LIN {X 0,Y 228.029,Z 967.337,A -85,B 0,C 180,E1 21811.233,E2 21811.233} C_VEL
LIN {X 0,Y 222.04,Z 977.557,A -85,B 0,C 180,E1 21813.343,E2 21813.343} C_VEL
LIN {X 0,Y 203.296,Z 1003.599,A -85,B 0,C 180,E1 21817.694,E2 21817.694} C_VEL
LIN {X 0,Y 184.311,Z 1025.745,A -85,B 0,C 180,E1 21824.225,E2 21824.225} C_VEL
LIN {X 0,Y 167.624,Z 1043.703,A -85,B 0,C 180,E1 21833.728,E2 21833.728} C_VEL
LIN {X 0,Y 157.775,Z 1054.755,A -85,B 0,C 180,E1 21844.418,E2 21844.418} C_VEL
LIN {X 0,Y 154.684,Z 1059.498,A -85,B 0,C 180,E1 21852.926,E2 21852.926} C_VEL
LIN {X 0,Y 154.96,Z 1063.359,A -85,B 0,C 180,E1 21867.202,E2 21867.202} C_VEL
LIN {X 0,Y 155.441,Z 1064.231,A -85,B 0,C 180,E1 21870.002,E2 21870.002} C_VEL
LIN {X 0,Y 154.103,Z 1063.62,A -85,B 0,C 180,E1 21881.334,E2 21881.334} C_VEL
LIN {X 0,Y 156.749,Z 1057.505,A -85,B 0,C 180,E1 21893.823,E2 21893.823} C_VEL
LIN {X 0,Y 166.557,Z 1045.003,A -85,B 0,C 180,E1 21905.9,E2 21905.9} C_VEL
LIN {X 0,Y 181.065,Z 1027.75,A -85,B 0,C 180,E1 21915.139,E2 21915.139} C_VEL
LIN {X 0,Y 197.137,Z 1006.697,A -85,B 0,C 180,E1 21921.789,E2 21921.789} C_VEL
LIN {X 0,Y 213.96,Z 980.35,A -85,B 0,C 180,E1 21926.713,E2 21926.713} C_VEL
LIN {X 0,Y 216.771,Z 975.207,A -85,B 0,C 180,E1 21927.424,E2 21927.424} C_VEL
LIN {X 0,Y 215.522,Z 959.866,A -85,B 0,C 180,E1 21933.374,E2 21933.374} C_VEL
LIN {X 0,Y 212.732,Z 946.935,A -85,B 0,C 180,E1 21940.342,E2 21940.342} C_VEL
LIN {X 0,Y 210.263,Z 938.618,A -85,B 0,C 180,E1 21947.476,E2 21947.476} C_VEL
LIN {X 0,Y 209.511,Z 933.278,A -85,B 0,C 180,E1 21955.804,E2 21955.804} C_VEL
LIN {X 0,Y 208.428,Z 937.644,A -85,B 0,C 180,E1 21964.111,E2 21964.111} C_VEL
LIN {X 0,Y 208.488,Z 945.436,A -85,B 0,C 180,E1 21971.461,E2 21971.461} C_VEL
LIN {X 0,Y 207.971,Z 957.227,A -85,B 0,C 180,E1 21978.834,E2 21978.834} C_VEL
LIN {X 0,Y 205.353,Z 971.666,A -85,B 0,C 180,E1 21986.184,E2 21986.184} C_VEL
LIN {X 0,Y 202.767,Z 979.395,A -85,B 0,C 180,E1 21989.847,E2 21989.847} C_VEL
LIN {X 0,Y 187.855,Z 996.811,A -85,B 0,C 180,E1 21996.292,E2 21996.292} C_VEL
LIN {X 0,Y 174.25,Z 1009.398,A -85,B 0,C 180,E1 22004.487,E2 22004.487} C_VEL
LIN {X 0,Y 164.735,Z 1016.233,A -85,B 0,C 180,E1 22013.313,E2 22013.313} C_VEL
LIN {X 0,Y 159.279,Z 1018.695,A -85,B 0,C 180,E1 22021.62,E2 22021.62} C_VEL
LIN {X 0,Y 156.492,Z 1018.02,A -85,B 0,C 180,E1 22029.898,E2 22029.898} C_VEL
LIN {X 0,Y 154.888,Z 1017.446,A -85,B 0,C 180,E1 22033.056,E2 22033.056} C_VEL
LIN {X 0,Y 149.377,Z 1013.798,A -85,B 0,C 180,E1 22041.859,E2 22041.859} C_VEL
LIN {X 0,Y 149.53,Z 1013.227,A -85,B 0,C 180,E1 22042.674,E2 22042.674} C_VEL
LIN {X 0,Y 155.199,Z 1001.57,A -85,B 0,C 180,E1 22054.194,E2 22054.194} C_VEL
LIN {X 0,Y 163.496,Z 986.022,A -85,B 0,C 180,E1 22063.22,E2 22063.22} C_VEL
LIN {X 0,Y 174.114,Z 964.454,A -85,B 0,C 180,E1 22071.019,E2 22071.019} C_VEL
LIN {X 0,Y 177.417,Z 956.35,A -85,B 0,C 180,E1 22073.245,E2 22073.245} C_VEL
LIN {X 0,Y 177.487,Z 938.518,A -85,B 0,C 180,E1 22079.2,E2 22079.2} C_VEL
LIN {X 0,Y 163.827,Z 940.595,A -85,B 0,C 180,E1 22083.878,E2 22083.878} C_VEL
LIN {X 0,Y 163.066,Z 940.258,A -85,B 0,C 180,E1 22084.495,E2 22084.495} C_VEL
LIN {X 0,Y 157.198,Z 966.499,A -85,B 0,C 180,E1 22090.811,E2 22090.811} C_VEL
LIN {X 0,Y 151.842,Z 988.828,A -85,B 0,C 180,E1 22099.154,E2 22099.154} C_VEL
LIN {X 0,Y 148.741,Z 1004.476,A -85,B 0,C 180,E1 22108.06,E2 22108.06} C_VEL
LIN {X 0,Y 148.185,Z 1016.057,A -85,B 0,C 180,E1 22118.312,E2 22118.312} C_VEL
LIN {X 0,Y 151.421,Z 1022.552,A -85,B 0,C 180,E1 22128.544,E2 22128.544} C_VEL
LIN {X 0,Y 155.312,Z 1024.197,A -85,B 0,C 180,E1 22134.48,E2 22134.48} C_VEL
LIN {X 0,Y 166.014,Z 1022.709,A -85,B 0,C 180,E1 22144.598,E2 22144.598} C_VEL
LIN {X 0,Y 180.205,Z 1015.966,A -85,B 0,C 180,E1 22153.03,E2 22153.03} C_VEL
LIN {X 0,Y 196.477,Z 1003.96,A -85,B 0,C 180,E1 22159.754,E2 22159.754} C_VEL
LIN {X 0,Y 214.009,Z 986.117,A -85,B 0,C 180,E1 22165.164,E2 22165.164} C_VEL
LIN {X 0,Y 220.51,Z 977.925,A -85,B 0,C 180,E1 22166.974,E2 22166.974} C_VEL
LIN {X 0,Y 222.968,Z 974.491,A -85,B 0,C 180,E1 22169.537,E2 22169.537} C_VEL
LIN {X 0,Y 222.507,Z 975.381,A -85,B 0,C 180,E1 22170.622,E2 22170.622} C_VEL
LIN {X 0,Y 215.741,Z 984.993,A -85,B 0,C 180,E1 22172.161,E2 22172.161} C_VEL
LIN {X 0,Y 194.53,Z 1010.583,A -85,B 0,C 180,E1 22177.084,E2 22177.084} C_VEL
LIN {X 0,Y 173.968,Z 1031.564,A -85,B 0,C 180,E1 22184.615,E2 22184.615} C_VEL
LIN {X 0,Y 157.729,Z 1046.889,A -85,B 0,C 180,E1 22194.836,E2 22194.836} C_VEL
LIN {X 0,Y 148.761,Z 1055.954,A -85,B 0,C 180,E1 22206.479,E2 22206.479} C_VEL
LIN {X 0,Y 146.505,Z 1059.588,A -85,B 0,C 180,E1 22218.074,E2 22218.074} C_VEL
LIN {X 0,Y 147.595,Z 1062.957,A -85,B 0,C 180,E1 22230.002,E2 22230.002} C_VEL
LIN {X 0,Y 146.253,Z 1062.469,A -85,B 0,C 180,E1 22241.952,E2 22241.952} C_VEL
LIN {X 0,Y 149.565,Z 1056.191,A -85,B 0,C 180,E1 22255.485,E2 22255.485} C_VEL
LIN {X 0,Y 160.402,Z 1043.804,A -85,B 0,C 180,E1 22267.849,E2 22267.849} C_VEL
LIN {X 0,Y 176.444,Z 1025.945,A -85,B 0,C 180,E1 22277.47,E2 22277.47} C_VEL
LIN {X 0,Y 193.605,Z 1004.417,A -85,B 0,C 180,E1 22284.083,E2 22284.083} C_VEL
LIN {X 0,Y 210.968,Z 977.854,A -85,B 0,C 180,E1 22288.843,E2 22288.843} C_VEL
LIN {X 0,Y 210.344,Z 964.721,A -85,B 0,C 180,E1 22294.366,E2 22294.366} C_VEL
LIN {X 0,Y 208.031,Z 951.826,A -85,B 0,C 180,E1 22301.908,E2 22301.908} C_VEL
LIN {X 0,Y 205.979,Z 944.435,A -85,B 0,C 180,E1 22309.361,E2 22309.361} C_VEL
LIN {X 0,Y 205.898,Z 940.4,A -85,B 0,C 180,E1 22315.731,E2 22315.731} C_VEL
LIN {X 0,Y 204.395,Z 944.731,A -85,B 0,C 180,E1 22324.192,E2 22324.192} C_VEL
LIN {X 0,Y 203.783,Z 952.605,A -85,B 0,C 180,E1 22331.683,E2 22331.683} C_VEL
LIN {X 0,Y 202.215,Z 964.628,A -85,B 0,C 180,E1 22339.392,E2 22339.392} C_VEL
LIN {X 0,Y 198.723,Z 977.474,A -85,B 0,C 180,E1 22346.237,E2 22346.237} C_VEL
LIN {X 0,Y 195.713,Z 983.429,A -85,B 0,C 180,E1 22348.932,E2 22348.932} C_VEL
LIN {X 0,Y 179.086,Z 1001.128,A -85,B 0,C 180,E1 22356.191,E2 22356.191} C_VEL
LIN {X 0,Y 165.411,Z 1012.493,A -85,B 0,C 180,E1 22364.814,E2 22364.814} C_VEL
LIN {X 0,Y 155.851,Z 1018.408,A -85,B 0,C 180,E1 22374.343,E2 22374.343} C_VEL
LIN {X 0,Y 149.602,Z 1019.899,A -85,B 0,C 180,E1 22386.117,E2 22386.117} C_VEL
LIN {X 0,Y 148.554,Z 1016.055,A -85,B 0,C 180,E1 22398.236,E2 22398.236} C_VEL
LIN {X 0,Y 149.53,Z 1013.227,A -85,B 0,C 180,E1 22402.674,E2 22402.674} C_VEL
LIN {X 0,Y 148.875,Z 1009.687,A -85,B 0,C 180,E1 22407.527,E2 22407.527} C_VEL
LIN {X 0,Y 147.619,Z 1003.02,A -85,B 0,C 180,E1 22414.754,E2 22414.754} C_VEL
LIN {X 0,Y 148.064,Z 1002.082,A -85,B 0,C 180,E1 22415.512,E2 22415.512} C_VEL
LIN {X 0,Y 157.724,Z 984.901,A -85,B 0,C 180,E1 22425.507,E2 22425.507} C_VEL
LIN {X 0,Y 168.707,Z 963.403,A -85,B 0,C 180,E1 22433.117,E2 22433.117} C_VEL
LIN {X 0,Y 170.899,Z 957.374,A -85,B 0,C 180,E1 22434.885,E2 22434.885} C_VEL
LIN {X 0,Y 170.904,Z 945.87,A -85,B 0,C 180,E1 22439.151,E2 22439.151} C_VEL
LIN {X 0,Y 161.241,Z 947.296,A -85,B 0,C 180,E1 22442.484,E2 22442.484} C_VEL
LIN {X 0,Y 155.877,Z 949.306,A -85,B 0,C 180,E1 22444.086,E2 22444.086} C_VEL
LIN {X 0,Y 153.649,Z 949.749,A -85,B 0,C 180,E1 22445.448,E2 22445.448} C_VEL
LIN {X 0,Y 147.267,Z 975.851,A -85,B 0,C 180,E1 22453.042,E2 22453.042} C_VEL
LIN {X 0,Y 142.62,Z 995.639,A -85,B 0,C 180,E1 22462.03,E2 22462.03} C_VEL
LIN {X 0,Y 140.25,Z 1010.132,A -85,B 0,C 180,E1 22472.02,E2 22472.02} C_VEL
LIN {X 0,Y 141.614,Z 1020.907,A -85,B 0,C 180,E1 22484.197,E2 22484.197} C_VEL
LIN {X 0,Y 146.983,Z 1025.26,A -85,B 0,C 180,E1 22494.166,E2 22494.166} C_VEL
LIN {X 0,Y 152.277,Z 1025.845,A -85,B 0,C 180,E1 22500.073,E2 22500.073} C_VEL
LIN {X 0,Y 166.607,Z 1022.246,A -85,B 0,C 180,E1 22510.535,E2 22510.535} C_VEL
LIN {X 0,Y 183.215,Z 1013.219,A -85,B 0,C 180,E1 22518.318,E2 22518.318} C_VEL
LIN {X 0,Y 202.615,Z 997.714,A -85,B 0,C 180,E1 22524.712,E2 22524.712} C_VEL
LIN {X 0,Y 216.289,Z 983.083,A -85,B 0,C 180,E1 22528.243,E2 22528.243} C_VEL
LIN {X 0,Y 217.862,Z 981.272,A -85,B 0,C 180,E1 22529.154,E2 22529.154} C_VEL
LIN {X 0,Y 216.382,Z 983.183,A -85,B 0,C 180,E1 22529.731,E2 22529.731} C_VEL
LIN {X 0,Y 194.367,Z 1008.192,A -85,B 0,C 180,E1 22534.143,E2 22534.143} C_VEL
LIN {X 0,Y 172.775,Z 1028.508,A -85,B 0,C 180,E1 22540.887,E2 22540.887} C_VEL
LIN {X 0,Y 154.561,Z 1043.785,A -85,B 0,C 180,E1 22550.453,E2 22550.453} C_VEL
LIN {X 0,Y 143.327,Z 1053.143,A -85,B 0,C 180,E1 22561.619,E2 22561.619} C_VEL
LIN {X 0,Y 139.345,Z 1057.074,A -85,B 0,C 180,E1 22570.978,E2 22570.978} C_VEL
LIN {X 0,Y 138.869,Z 1058.428,A -85,B 0,C 180,E1 22581.609,E2 22581.609} C_VEL
LIN {X 0,Y 139.755,Z 1061.663,A -85,B 0,C 180,E1 22590.002,E2 22590.002} C_VEL
LIN {X 0,Y 138.392,Z 1061.312,A -85,B 0,C 180,E1 22602.641,E2 22602.641} C_VEL
LIN {X 0,Y 142.279,Z 1055.149,A -85,B 0,C 180,E1 22616.892,E2 22616.892} C_VEL
LIN {X 0,Y 154.065,Z 1042.938,A -85,B 0,C 180,E1 22629.704,E2 22629.704} C_VEL
LIN {X 0,Y 170.283,Z 1026.144,A -85,B 0,C 180,E1 22639.096,E2 22639.096} C_VEL
LIN {X 0,Y 189.151,Z 1003.779,A -85,B 0,C 180,E1 22646.081,E2 22646.081} C_VEL
LIN {X 0,Y 205.232,Z 980.507,A -85,B 0,C 180,E1 22650.343,E2 22650.343} C_VEL
LIN {X 0,Y 204.846,Z 967.229,A -85,B 0,C 180,E1 22656.543,E2 22656.543} C_VEL
LIN {X 0,Y 203.246,Z 956.398,A -85,B 0,C 180,E1 22663.73,E2 22663.73} C_VEL
LIN {X 0,Y 201.732,Z 950.029,A -85,B 0,C 180,E1 22671.315,E2 22671.315} C_VEL
LIN {X 0,Y 201.977,Z 947.406,A -85,B 0,C 180,E1 22675.648,E2 22675.648} C_VEL
LIN {X 0,Y 200.398,Z 950.179,A -85,B 0,C 180,E1 22682.109,E2 22682.109} C_VEL
LIN {X 0,Y 199.376,Z 956.143,A -85,B 0,C 180,E1 22689.157,E2 22689.157} C_VEL
LIN {X 0,Y 197.202,Z 967.09,A -85,B 0,C 180,E1 22697.111,E2 22697.111} C_VEL
LIN {X 0,Y 193.399,Z 979.33,A -85,B 0,C 180,E1 22704.201,E2 22704.201} C_VEL
LIN {X 0,Y 191.142,Z 984.423,A -85,B 0,C 180,E1 22706.977,E2 22706.977} C_VEL
LIN {X 0,Y 174.334,Z 1001.641,A -85,B 0,C 180,E1 22713.998,E2 22713.998} C_VEL
LIN {X 0,Y 159.666,Z 1013.238,A -85,B 0,C 180,E1 22722.697,E2 22722.697} C_VEL
LIN {X 0,Y 149.196,Z 1019.423,A -85,B 0,C 180,E1 22732.488,E2 22732.488} C_VEL
LIN {X 0,Y 142.17,Z 1021.163,A -85,B 0,C 180,E1 22744.784,E2 22744.784} C_VEL
LIN {X 0,Y 140.634,Z 1017.58,A -85,B 0,C 180,E1 22757.563,E2 22757.563} C_VEL
LIN {X 0,Y 144.696,Z 1008.44,A -85,B 0,C 180,E1 22769.998,E2 22769.998} C_VEL
LIN {X 0,Y 148.064,Z 1002.082,A -85,B 0,C 180,E1 22775.512,E2 22775.512} C_VEL
LIN {X 0,Y 147.385,Z 997.386,A -85,B 0,C 180,E1 22779.727,E2 22779.727} C_VEL
LIN {X 0,Y 147.297,Z 992.02,A -85,B 0,C 180,E1 22783.836,E2 22783.836} C_VEL
LIN {X 0,Y 158.653,Z 971.863,A -85,B 0,C 180,E1 22792.439,E2 22792.439} C_VEL
LIN {X 0,Y 164.249,Z 960.2,A -85,B 0,C 180,E1 22795.966,E2 22795.966} C_VEL
LIN {X 0,Y 165.075,Z 952.705,A -85,B 0,C 180,E1 22798.78,E2 22798.78} C_VEL
LIN {X 0,Y 152.734,Z 955.58,A -85,B 0,C 180,E1 22802.756,E2 22802.756} C_VEL
LIN {X 0,Y 145.006,Z 957.339,A -85,B 0,C 180,E1 22805.811,E2 22805.811} C_VEL
LIN {X 0,Y 143.906,Z 959.455,A -85,B 0,C 180,E1 22806.868,E2 22806.868} C_VEL
LIN {X 0,Y 137.626,Z 983.982,A -85,B 0,C 180,E1 22815.55,E2 22815.55} C_VEL
LIN {X 0,Y 133.503,Z 1002.243,A -85,B 0,C 180,E1 22825.573,E2 22825.573} C_VEL
LIN {X 0,Y 132.268,Z 1015.032,A -85,B 0,C 180,E1 22836.309,E2 22836.309} C_VEL
LIN {X 0,Y 134.774,Z 1023.078,A -85,B 0,C 180,E1 22847.106,E2 22847.106} C_VEL
LIN {X 0,Y 138.569,Z 1026.061,A -85,B 0,C 180,E1 22853.81,E2 22853.81} C_VEL
LIN {X 0,Y 150.685,Z 1026.951,A -85,B 0,C 180,E1 22865.838,E2 22865.838} C_VEL
LIN {X 0,Y 165.335,Z 1022.545,A -85,B 0,C 180,E1 22874.598,E2 22874.598} C_VEL
LIN {X 0,Y 183.447,Z 1012.761,A -85,B 0,C 180,E1 22881.858,E2 22881.858} C_VEL
LIN {X 0,Y 202.545,Z 997.761,A -85,B 0,C 180,E1 22887.41,E2 22887.41} C_VEL
LIN {X 0,Y 207.432,Z 993.164,A -85,B 0,C 180,E1 22888.851,E2 22888.851} C_VEL
LIN {X 0,Y 182.769,Z 1016.977,A -85,B 0,C 180,E1 22894.067,E2 22894.067} C_VEL
LIN {X 0,Y 161.491,Z 1034.127,A -85,B 0,C 180,E1 22901.408,E2 22901.408} C_VEL
LIN {X 0,Y 143.469,Z 1047.146,A -85,B 0,C 180,E1 22912.252,E2 22912.252} C_VEL
LIN {X 0,Y 133.19,Z 1054.601,A -85,B 0,C 180,E1 22925.572,E2 22925.572} C_VEL
LIN {X 0,Y 131.057,Z 1057.283,A -85,B 0,C 180,E1 22941.64,E2 22941.64} C_VEL
LIN {X 0,Y 131.933,Z 1060.373,A -85,B 0,C 180,E1 22950.002,E2 22950.002} C_VEL
LIN {X 0,Y 130.575,Z 1060.156,A -85,B 0,C 180,E1 22963.412,E2 22963.412} C_VEL
LIN {X 0,Y 134.172,Z 1055.063,A -85,B 0,C 180,E1 22976.835,E2 22976.835} C_VEL
LIN {X 0,Y 146.125,Z 1043.754,A -85,B 0,C 180,E1 22990.363,E2 22990.363} C_VEL
LIN {X 0,Y 163.909,Z 1026.724,A -85,B 0,C 180,E1 23000.683,E2 23000.683} C_VEL
LIN {X 0,Y 183.386,Z 1005.118,A -85,B 0,C 180,E1 23007.733,E2 23007.733} C_VEL
LIN {X 0,Y 199.357,Z 983.496,A -85,B 0,C 180,E1 23011.835,E2 23011.835} C_VEL
LIN {X 0,Y 199.558,Z 971.859,A -85,B 0,C 180,E1 23017.656,E2 23017.656} C_VEL
LIN {X 0,Y 198.579,Z 962.28,A -85,B 0,C 180,E1 23024.471,E2 23024.471} C_VEL
LIN {X 0,Y 197.643,Z 954.687,A -85,B 0,C 180,E1 23034.82,E2 23034.82} C_VEL
LIN {X 0,Y 196.526,Z 955.593,A -85,B 0,C 180,E1 23039.944,E2 23039.944} C_VEL
LIN {X 0,Y 194.441,Z 962.436,A -85,B 0,C 180,E1 23048.898,E2 23048.898} C_VEL
LIN {X 0,Y 191.799,Z 971.74,A -85,B 0,C 180,E1 23056.094,E2 23056.094} C_VEL
LIN {X 0,Y 187.488,Z 982.869,A -85,B 0,C 180,E1 23063.042,E2 23063.042} C_VEL
LIN {X 0,Y 184.832,Z 987.642,A -85,B 0,C 180,E1 23065.695,E2 23065.695} C_VEL
LIN {X 0,Y 166.835,Z 1004.649,A -85,B 0,C 180,E1 23073.103,E2 23073.103} C_VEL
LIN {X 0,Y 150.501,Z 1016.3,A -85,B 0,C 180,E1 23083.163,E2 23083.163} C_VEL
LIN {X 0,Y 142.725,Z 1020.435,A -85,B 0,C 180,E1 23090.466,E2 23090.466} C_VEL
LIN {X 0,Y 134.571,Z 1022.36,A -85,B 0,C 180,E1 23103.931,E2 23103.931} C_VEL
LIN {X 0,Y 132.751,Z 1019.042,A -85,B 0,C 180,E1 23116.812,E2 23116.812} C_VEL
LIN {X 0,Y 136.703,Z 1010.183,A -85,B 0,C 180,E1 23129.998,E2 23129.998} C_VEL
LIN {X 0,Y 144.762,Z 996.321,A -85,B 0,C 180,E1 23141.307,E2 23141.307} C_VEL
LIN {X 0,Y 147.297,Z 992.02,A -85,B 0,C 180,E1 23143.836,E2 23143.836} C_VEL
LIN {X 0,Y 149.883,Z 982.506,A -85,B 0,C 180,E1 23149.419,E2 23149.419} C_VEL
LIN {X 0,Y 152.958,Z 971.748,A -85,B 0,C 180,E1 23154.546,E2 23154.546} C_VEL
LIN {X 0,Y 158.067,Z 960.594,A -85,B 0,C 180,E1 23158.117,E2 23158.117} C_VEL
LIN {X 0,Y 158.278,Z 959.448,A -85,B 0,C 180,E1 23158.572,E2 23158.572} C_VEL
LIN {X 0,Y 138.692,Z 964.583,A -85,B 0,C 180,E1 23165.213,E2 23165.213} C_VEL
LIN {X 0,Y 134.955,Z 965.203,A -85,B 0,C 180,E1 23167.555,E2 23167.555} C_VEL
LIN {X 0,Y 128.999,Z 987.722,A -85,B 0,C 180,E1 23176.536,E2 23176.536} C_VEL
LIN {X 0,Y 124.976,Z 1006.133,A -85,B 0,C 180,E1 23187.996,E2 23187.996} C_VEL
LIN {X 0,Y 124.791,Z 1018.676,A -85,B 0,C 180,E1 23200.228,E2 23200.228} C_VEL
LIN {X 0,Y 130.146,Z 1026.576,A -85,B 0,C 180,E1 23213.408,E2 23213.408} C_VEL
LIN {X 0,Y 142.495,Z 1028.813,A -85,B 0,C 180,E1 23226.175,E2 23226.175} C_VEL
LIN {X 0,Y 156.657,Z 1025.904,A -85,B 0,C 180,E1 23234.882,E2 23234.882} C_VEL
LIN {X 0,Y 176.323,Z 1017.193,A -85,B 0,C 180,E1 23242.854,E2 23242.854} C_VEL
LIN {X 0,Y 195.416,Z 1004.39,A -85,B 0,C 180,E1 23248.282,E2 23248.282} C_VEL
LIN {X 0,Y 168.399,Z 1026.15,A -85,B 0,C 180,E1 23254.875,E2 23254.875} C_VEL
LIN {X 0,Y 146.792,Z 1040.697,A -85,B 0,C 180,E1 23263.782,E2 23263.782} C_VEL
LIN {X 0,Y 131.981,Z 1049.734,A -85,B 0,C 180,E1 23275.001,E2 23275.001} C_VEL
LIN {X 0,Y 124.221,Z 1054.414,A -85,B 0,C 180,E1 23288.555,E2 23288.555} C_VEL
LIN {X 0,Y 123.246,Z 1055.205,A -85,B 0,C 180,E1 23299.72,E2 23299.72} C_VEL
LIN {X 0,Y 124.106,Z 1059.083,A -85,B 0,C 180,E1 23310.002,E2 23310.002} C_VEL
LIN {X 0,Y 122.766,Z 1058.971,A -85,B 0,C 180,E1 23324.283,E2 23324.283} C_VEL
LIN {X 0,Y 126.979,Z 1054.032,A -85,B 0,C 180,E1 23338.489,E2 23338.489} C_VEL
LIN {X 0,Y 140.052,Z 1042.895,A -85,B 0,C 180,E1 23352.51,E2 23352.51} C_VEL
LIN {X 0,Y 158.931,Z 1026.054,A -85,B 0,C 180,E1 23362.929,E2 23362.929} C_VEL
LIN {X 0,Y 179.345,Z 1004.546,A -85,B 0,C 180,E1 23369.924,E2 23369.924} C_VEL
LIN {X 0,Y 193.251,Z 986.794,A -85,B 0,C 180,E1 23373.352,E2 23373.352} C_VEL
LIN {X 0,Y 194.165,Z 978.377,A -85,B 0,C 180,E1 23377.606,E2 23377.606} C_VEL
LIN {X 0,Y 193.709,Z 968.016,A -85,B 0,C 180,E1 23385.231,E2 23385.231} C_VEL
LIN {X 0,Y 193.253,Z 960.939,A -85,B 0,C 180,E1 23395.451,E2 23395.451} C_VEL
LIN {X 0,Y 191.151,Z 963.426,A -85,B 0,C 180,E1 23402.211,E2 23402.211} C_VEL
LIN {X 0,Y 189.072,Z 969.071,A -85,B 0,C 180,E1 23409.153,E2 23409.153} C_VEL
LIN {X 0,Y 185.44,Z 978.512,A -85,B 0,C 180,E1 23416.661,E2 23416.661} C_VEL
LIN {X 0,Y 179.534,Z 989.844,A -85,B 0,C 180,E1 23423.956,E2 23423.956} C_VEL
LIN {X 0,Y 161.766,Z 1005.771,A -85,B 0,C 180,E1 23430.995,E2 23430.995} C_VEL
LIN {X 0,Y 144.843,Z 1017.198,A -85,B 0,C 180,E1 23440.853,E2 23440.853} C_VEL
LIN {X 0,Y 132.538,Z 1022.819,A -85,B 0,C 180,E1 23452.925,E2 23452.925} C_VEL
LIN {X 0,Y 127.549,Z 1023.61,A -85,B 0,C 180,E1 23461.649,E2 23461.649} C_VEL
LIN {X 0,Y 124.867,Z 1020.5,A -85,B 0,C 180,E1 23475.963,E2 23475.963} C_VEL
LIN {X 0,Y 128.692,Z 1011.925,A -85,B 0,C 180,E1 23489.998,E2 23489.998} C_VEL
LIN {X 0,Y 137.734,Z 997.286,A -85,B 0,C 180,E1 23502.698,E2 23502.698} C_VEL
LIN {X 0,Y 149.459,Z 977.971,A -85,B 0,C 180,E1 23512.325,E2 23512.325} C_VEL
LIN {X 0,Y 152.958,Z 971.748,A -85,B 0,C 180,E1 23514.546,E2 23514.546} C_VEL
LIN {X 0,Y 152.567,Z 968.801,A -85,B 0,C 180,E1 23516.328,E2 23516.328} C_VEL
LIN {X 0,Y 146.457,Z 967.65,A -85,B 0,C 180,E1 23519.581,E2 23519.581} C_VEL
LIN {X 0,Y 130.899,Z 971.037,A -85,B 0,C 180,E1 23525.587,E2 23525.587} C_VEL
LIN {X 0,Y 125.47,Z 972.244,A -85,B 0,C 180,E1 23528.957,E2 23528.957} C_VEL
LIN {X 0,Y 119.632,Z 994.25,A -85,B 0,C 180,E1 23539.404,E2 23539.404} C_VEL
LIN {X 0,Y 116.541,Z 1011.595,A -85,B 0,C 180,E1 23552.413,E2 23552.413} C_VEL
LIN {X 0,Y 118.821,Z 1023.708,A -85,B 0,C 180,E1 23567.217,E2 23567.217} C_VEL
LIN {X 0,Y 127.173,Z 1029.413,A -85,B 0,C 180,E1 23580.087,E2 23580.087} C_VEL
LIN {X 0,Y 142.698,Z 1029.846,A -85,B 0,C 180,E1 23592.326,E2 23592.326} C_VEL
LIN {X 0,Y 163.175,Z 1023.959,A -85,B 0,C 180,E1 23601.85,E2 23601.85} C_VEL
LIN {X 0,Y 182.474,Z 1014.154,A -85,B 0,C 180,E1 23607.808,E2 23607.808} C_VEL
LIN {X 0,Y 154.125,Z 1033.298,A -85,B 0,C 180,E1 23615.863,E2 23615.863} C_VEL
LIN {X 0,Y 132.618,Z 1045.282,A -85,B 0,C 180,E1 23626.767,E2 23626.767} C_VEL
LIN {X 0,Y 120.089,Z 1051.454,A -85,B 0,C 180,E1 23639.717,E2 23639.717} C_VEL
LIN {X 0,Y 115.435,Z 1053.768,A -85,B 0,C 180,E1 23659.016,E2 23659.016} C_VEL
LIN {X 0,Y 116.243,Z 1057.776,A -85,B 0,C 180,E1 23670.003,E2 23670.003} C_VEL
LIN {X 0,Y 114.997,Z 1057.775,A -85,B 0,C 180,E1 23685.27,E2 23685.27} C_VEL
LIN {X 0,Y 119.913,Z 1053.002,A -85,B 0,C 180,E1 23700.338,E2 23700.338} C_VEL
LIN {X 0,Y 134.183,Z 1042.019,A -85,B 0,C 180,E1 23714.851,E2 23714.851} C_VEL
LIN {X 0,Y 154.189,Z 1025.383,A -85,B 0,C 180,E1 23725.328,E2 23725.328} C_VEL
LIN {X 0,Y 175.46,Z 1004.082,A -85,B 0,C 180,E1 23732.193,E2 23732.193} C_VEL
LIN {X 0,Y 187.382,Z 989.809,A -85,B 0,C 180,E1 23734.984,E2 23734.984} C_VEL
LIN {X 0,Y 188.486,Z 984.741,A -85,B 0,C 180,E1 23737.484,E2 23737.484} C_VEL
LIN {X 0,Y 188.712,Z 975.319,A -85,B 0,C 180,E1 23744.326,E2 23744.326} C_VEL
LIN {X 0,Y 188.227,Z 968.687,A -85,B 0,C 180,E1 23753.014,E2 23753.014} C_VEL
LIN {X 0,Y 188.466,Z 967.417,A -85,B 0,C 180,E1 23755.335,E2 23755.335} C_VEL
LIN {X 0,Y 186.092,Z 969.785,A -85,B 0,C 180,E1 23762.271,E2 23762.271} C_VEL
LIN {X 0,Y 183.359,Z 975.524,A -85,B 0,C 180,E1 23769.44,E2 23769.44} C_VEL
LIN {X 0,Y 178.75,Z 984.72,A -85,B 0,C 180,E1 23776.936,E2 23776.936} C_VEL
LIN {X 0,Y 174.361,Z 991.929,A -85,B 0,C 180,E1 23781.92,E2 23781.92} C_VEL
LIN {X 0,Y 156.033,Z 1007.554,A -85,B 0,C 180,E1 23789.149,E2 23789.149} C_VEL
LIN {X 0,Y 137.652,Z 1019.046,A -85,B 0,C 180,E1 23799.647,E2 23799.647} C_VEL
LIN {X 0,Y 124.62,Z 1024.269,A -85,B 0,C 180,E1 23812.589,E2 23812.589} C_VEL
LIN {X 0,Y 117.791,Z 1024.046,A -85,B 0,C 180,E1 23827.315,E2 23827.315} C_VEL
LIN {X 0,Y 118,Z 1018.524,A -85,B 0,C 180,E1 23842.625,E2 23842.625} C_VEL
LIN {X 0,Y 124.668,Z 1007.356,A -85,B 0,C 180,E1 23856.973,E2 23856.973} C_VEL
LIN {X 0,Y 135.492,Z 991.218,A -85,B 0,C 180,E1 23868.472,E2 23868.472} C_VEL
LIN {X 0,Y 148.358,Z 970.014,A -85,B 0,C 180,E1 23877.319,E2 23877.319} C_VEL
LIN {X 0,Y 150.004,Z 967.156,A -85,B 0,C 180,E1 23878.192,E2 23878.192} C_VEL
LIN {X 0,Y 147.276,Z 967.341,A -85,B 0,C 180,E1 23879.29,E2 23879.29} C_VEL
LIN {X 0,Y 130.899,Z 971.037,A -85,B 0,C 180,E1 23885.587,E2 23885.587} C_VEL
LIN {X 0,Y 121.588,Z 975.266,A -85,B 0,C 180,E1 23888.718,E2 23888.718} C_VEL
LIN {X 0,Y 115.514,Z 980.97,A -85,B 0,C 180,E1 23891.588,E2 23891.588} C_VEL
LIN {X 0,Y 115.134,Z 981.973,A -85,B 0,C 180,E1 23892.078,E2 23892.078} C_VEL
LIN {X 0,Y 110.009,Z 1002.178,A -85,B 0,C 180,E1 23904.191,E2 23904.191} C_VEL
LIN {X 0,Y 108.657,Z 1016.609,A -85,B 0,C 180,E1 23917.589,E2 23917.589} C_VEL
LIN {X 0,Y 113.236,Z 1026.743,A -85,B 0,C 180,E1 23932.418,E2 23932.418} C_VEL
LIN {X 0,Y 125.938,Z 1031.738,A -85,B 0,C 180,E1 23946.991,E2 23946.991} C_VEL
LIN {X 0,Y 144.626,Z 1030.42,A -85,B 0,C 180,E1 23958.377,E2 23958.377} C_VEL
LIN {X 0,Y 165.119,Z 1023.926,A -85,B 0,C 180,E1 23966.072,E2 23966.072} C_VEL
LIN {X 0,Y 169.419,Z 1022.041,A -85,B 0,C 180,E1 23967.318,E2 23967.318} C_VEL
LIN {X 0,Y 163.822,Z 1025.642,A -85,B 0,C 180,E1 23969.215,E2 23969.215} C_VEL
LIN {X 0,Y 138.347,Z 1039.394,A -85,B 0,C 180,E1 23977.896,E2 23977.896} C_VEL
LIN {X 0,Y 119.101,Z 1047.95,A -85,B 0,C 180,E1 23990.537,E2 23990.537} C_VEL
LIN {X 0,Y 109.428,Z 1051.458,A -85,B 0,C 180,E1 24005.478,E2 24005.478} C_VEL
LIN {X 0,Y 107.767,Z 1051.574,A -85,B 0,C 180,E1 24016.712,E2 24016.712} C_VEL
LIN {X 0,Y 108.404,Z 1056.474,A -85,B 0,C 180,E1 24030.003,E2 24030.003} C_VEL
LIN {X 0,Y 107.267,Z 1056.579,A -85,B 0,C 180,E1 24046.401,E2 24046.401} C_VEL
LIN {X 0,Y 112.983,Z 1051.962,A -85,B 0,C 180,E1 24062.418,E2 24062.418} C_VEL
LIN {X 0,Y 128.542,Z 1041.143,A -85,B 0,C 180,E1 24077.41,E2 24077.41} C_VEL
LIN {X 0,Y 149.758,Z 1024.705,A -85,B 0,C 180,E1 24087.861,E2 24087.861} C_VEL
LIN {X 0,Y 171.866,Z 1003.618,A -85,B 0,C 180,E1 24094.558,E2 24094.558} C_VEL
LIN {X 0,Y 182.432,Z 991.181,A -85,B 0,C 180,E1 24097.165,E2 24097.165} C_VEL
LIN {X 0,Y 183.332,Z 981.954,A -85,B 0,C 180,E1 24103.853,E2 24103.853} C_VEL
LIN {X 0,Y 183.166,Z 976.388,A -85,B 0,C 180,E1 24110.427,E2 24110.427} C_VEL
LIN {X 0,Y 183.409,Z 973.696,A -85,B 0,C 180,E1 24115.206,E2 24115.206} C_VEL
LIN {X 0,Y 180.871,Z 975.793,A -85,B 0,C 180,E1 24122.096,E2 24122.096} C_VEL
LIN {X 0,Y 177.263,Z 981.814,A -85,B 0,C 180,E1 24129.768,E2 24129.768} C_VEL
LIN {X 0,Y 172.484,Z 989.573,A -85,B 0,C 180,E1 24136.377,E2 24136.377} C_VEL
LIN {X 0,Y 168.492,Z 995.06,A -85,B 0,C 180,E1 24140.445,E2 24140.445} C_VEL
LIN {X 0,Y 149.494,Z 1010.031,A -85,B 0,C 180,E1 24147.596,E2 24147.596} C_VEL
LIN {X 0,Y 132.523,Z 1019.881,A -85,B 0,C 180,E1 24156.89,E2 24156.89} C_VEL
LIN {X 0,Y 118.163,Z 1025.352,A -85,B 0,C 180,E1 24170.155,E2 24170.155} C_VEL
LIN {X 0,Y 110.314,Z 1025.367,A -85,B 0,C 180,E1 24185.682,E2 24185.682} C_VEL
LIN {X 0,Y 109.993,Z 1020.105,A -85,B 0,C 180,E1 24202.085,E2 24202.085} C_VEL
LIN {X 0,Y 116.785,Z 1009.231,A -85,B 0,C 180,E1 24217.447,E2 24217.447} C_VEL
LIN {X 0,Y 127.684,Z 993.905,A -85,B 0,C 180,E1 24229.371,E2 24229.371} C_VEL
LIN {X 0,Y 139.59,Z 975.829,A -85,B 0,C 180,E1 24237.687,E2 24237.687} C_VEL
LIN {X 0,Y 139.929,Z 974.072,A -85,B 0,C 180,E1 24238.673,E2 24238.673} C_VEL
LIN {X 0,Y 116.078,Z 978.546,A -85,B 0,C 180,E1 24250.501,E2 24250.501} C_VEL
LIN {X 0,Y 115.134,Z 981.973,A -85,B 0,C 180,E1 24252.078,E2 24252.078} C_VEL
LIN {X 0,Y 110.282,Z 990.768,A -85,B 0,C 180,E1 24256.428,E2 24256.428} C_VEL
LIN {X 0,Y 102.196,Z 1002.375,A -85,B 0,C 180,E1 24263.966,E2 24263.966} C_VEL
LIN {X 0,Y 101.873,Z 1003.631,A -85,B 0,C 180,E1 24264.96,E2 24264.96} C_VEL
LIN {X 0,Y 101.161,Z 1019.001,A -85,B 0,C 180,E1 24280.728,E2 24280.728} C_VEL
LIN {X 0,Y 108.188,Z 1029.283,A -85,B 0,C 180,E1 24297.505,E2 24297.505} C_VEL
LIN {X 0,Y 123.934,Z 1033.464,A -85,B 0,C 180,E1 24312.23,E2 24312.23} C_VEL
LIN {X 0,Y 142.482,Z 1031.901,A -85,B 0,C 180,E1 24321.908,E2 24321.908} C_VEL
LIN {X 0,Y 156.202,Z 1028.324,A -85,B 0,C 180,E1 24326.81,E2 24326.81} C_VEL
LIN {X 0,Y 156.491,Z 1028.472,A -85,B 0,C 180,E1 24327.653,E2 24327.653} C_VEL
LIN {X 0,Y 128.702,Z 1041.222,A -85,B 0,C 180,E1 24337.435,E2 24337.435} C_VEL
LIN {X 0,Y 112.997,Z 1046.956,A -85,B 0,C 180,E1 24347.94,E2 24347.94} C_VEL
LIN {X 0,Y 102.193,Z 1049.828,A -85,B 0,C 180,E1 24363.614,E2 24363.614} C_VEL
LIN {X 0,Y 100.175,Z 1049.615,A -85,B 0,C 180,E1 24374.666,E2 24374.666} C_VEL
LIN {X 0,Y 100.533,Z 1055.17,A -85,B 0,C 180,E1 24390.003,E2 24390.003} C_VEL
LIN {X 0,Y 99.571,Z 1055.383,A -85,B 0,C 180,E1 24407.708,E2 24407.708} C_VEL
LIN {X 0,Y 106.235,Z 1050.902,A -85,B 0,C 180,E1 24424.76,E2 24424.76} C_VEL
LIN {X 0,Y 123.188,Z 1040.266,A -85,B 0,C 180,E1 24440.194,E2 24440.194} C_VEL
LIN {X 0,Y 145.637,Z 1024.026,A -85,B 0,C 180,E1 24450.543,E2 24450.543} C_VEL
LIN {X 0,Y 168.504,Z 1003.238,A -85,B 0,C 180,E1 24456.998,E2 24456.998} C_VEL
LIN {X 0,Y 176.017,Z 995.208,A -85,B 0,C 180,E1 24458.576,E2 24458.576} C_VEL
LIN {X 0,Y 177.614,Z 987.993,A -85,B 0,C 180,E1 24463.746,E2 24463.746} C_VEL
LIN {X 0,Y 177.823,Z 982.505,A -85,B 0,C 180,E1 24470.136,E2 24470.136} C_VEL
LIN {X 0,Y 178.092,Z 979.771,A -85,B 0,C 180,E1 24475.063,E2 24475.063} C_VEL
LIN {X 0,Y 175.146,Z 981.901,A -85,B 0,C 180,E1 24482.413,E2 24482.413} C_VEL
LIN {X 0,Y 170.786,Z 987.911,A -85,B 0,C 180,E1 24490.142,E2 24490.142} C_VEL
LIN {X 0,Y 164.075,Z 996.63,A -85,B 0,C 180,E1 24497.733,E2 24497.733} C_VEL
LIN {X 0,Y 160.56,Z 999.903,A -85,B 0,C 180,E1 24499.433,E2 24499.433} C_VEL
LIN {X 0,Y 139.961,Z 1014.296,A -85,B 0,C 180,E1 24507.307,E2 24507.307} C_VEL
LIN {X 0,Y 121.34,Z 1023.485,A -85,B 0,C 180,E1 24518.465,E2 24518.465} C_VEL
LIN {X 0,Y 111.979,Z 1026.434,A -85,B 0,C 180,E1 24527.46,E2 24527.46} C_VEL
LIN {X 0,Y 102.944,Z 1026.693,A -85,B 0,C 180,E1 24543.814,E2 24543.814} C_VEL
LIN {X 0,Y 101.99,Z 1021.679,A -85,B 0,C 180,E1 24561.46,E2 24561.46} C_VEL
LIN {X 0,Y 108.897,Z 1011.081,A -85,B 0,C 180,E1 24577.989,E2 24577.989} C_VEL
LIN {X 0,Y 120.843,Z 995.291,A -85,B 0,C 180,E1 24591.111,E2 24591.111} C_VEL
LIN {X 0,Y 130.928,Z 981.073,A -85,B 0,C 180,E1 24598.224,E2 24598.224} C_VEL
LIN {X 0,Y 123.96,Z 981.85,A -85,B 0,C 180,E1 24601.453,E2 24601.453} C_VEL
LIN {X 0,Y 107.138,Z 984.454,A -85,B 0,C 180,E1 24611.777,E2 24611.777} C_VEL
LIN {X 0,Y 101.873,Z 1003.631,A -85,B 0,C 180,E1 24624.96,E2 24624.96} C_VEL
LIN {X 0,Y 98.433,Z 1010.56,A -85,B 0,C 180,E1 24631.027,E2 24631.027} C_VEL
LIN {X 0,Y 93.435,Z 1019.167,A -85,B 0,C 180,E1 24641.342,E2 24641.342} C_VEL
LIN {X 0,Y 93.539,Z 1020.045,A -85,B 0,C 180,E1 24642.577,E2 24642.577} C_VEL
LIN {X 0,Y 101.634,Z 1030.388,A -85,B 0,C 180,E1 24660.109,E2 24660.109} C_VEL
LIN {X 0,Y 118.439,Z 1034.958,A -85,B 0,C 180,E1 24674.904,E2 24674.904} C_VEL
LIN {X 0,Y 140.929,Z 1033.433,A -85,B 0,C 180,E1 24685.527,E2 24685.527} C_VEL
LIN {X 0,Y 144.102,Z 1032.815,A -85,B 0,C 180,E1 24686.654,E2 24686.654} C_VEL
LIN {X 0,Y 141.254,Z 1034.228,A -85,B 0,C 180,E1 24688.086,E2 24688.086} C_VEL
LIN {X 0,Y 116.192,Z 1043.261,A -85,B 0,C 180,E1 24698.574,E2 24698.574} C_VEL
LIN {X 0,Y 99.99,Z 1047.464,A -85,B 0,C 180,E1 24712.725,E2 24712.725} C_VEL
LIN {X 0,Y 92.506,Z 1048.107,A -85,B 0,C 180,E1 24733.359,E2 24733.359} C_VEL
LIN {X 0,Y 92.676,Z 1053.868,A -85,B 0,C 180,E1 24750.003,E2 24750.003} C_VEL
LIN {X 0,Y 91.93,Z 1054.188,A -85,B 0,C 180,E1 24769.236,E2 24769.236} C_VEL
LIN {X 0,Y 99.672,Z 1049.839,A -85,B 0,C 180,E1 24787.422,E2 24787.422} C_VEL
LIN {X 0,Y 118.154,Z 1039.389,A -85,B 0,C 180,E1 24803.22,E2 24803.22} C_VEL
LIN {X 0,Y 141.829,Z 1023.347,A -85,B 0,C 180,E1 24813.393,E2 24813.393} C_VEL
LIN {X 0,Y 166.4,Z 1001.975,A -85,B 0,C 180,E1 24819.714,E2 24819.714} C_VEL
LIN {X 0,Y 170.122,Z 998.221,A -85,B 0,C 180,E1 24820.445,E2 24820.445} C_VEL
LIN {X 0,Y 171.556,Z 994.282,A -85,B 0,C 180,E1 24823.156,E2 24823.156} C_VEL
LIN {X 0,Y 172.203,Z 988.431,A -85,B 0,C 180,E1 24829.811,E2 24829.811} C_VEL
LIN {X 0,Y 172.55,Z 985.604,A -85,B 0,C 180,E1 24834.904,E2 24834.904} C_VEL
LIN {X 0,Y 170.625,Z 986.45,A -85,B 0,C 180,E1 24839.935,E2 24839.935} C_VEL
LIN {X 0,Y 166.065,Z 991.235,A -85,B 0,C 180,E1 24847.787,E2 24847.787} C_VEL
LIN {X 0,Y 160.122,Z 998.045,A -85,B 0,C 180,E1 24854.547,E2 24854.547} C_VEL
LIN {X 0,Y 156.528,Z 1001.494,A -85,B 0,C 180,E1 24857.049,E2 24857.049} C_VEL
LIN {X 0,Y 133.966,Z 1016.294,A -85,B 0,C 180,E1 24865.285,E2 24865.285} C_VEL
LIN {X 0,Y 113.919,Z 1025.264,A -85,B 0,C 180,E1 24877.109,E2 24877.109} C_VEL
LIN {X 0,Y 99.9,Z 1028.422,A -85,B 0,C 180,E1 24892.678,E2 24892.678} C_VEL
LIN {X 0,Y 93.681,Z 1026.263,A -85,B 0,C 180,E1 24911.138,E2 24911.138} C_VEL
LIN {X 0,Y 96.608,Z 1018.738,A -85,B 0,C 180,E1 24929.997,E2 24929.997} C_VEL
LIN {X 0,Y 106.973,Z 1005.453,A -85,B 0,C 180,E1 24946.441,E2 24946.441} C_VEL
LIN {X 0,Y 120.75,Z 988.101,A -85,B 0,C 180,E1 24957.828,E2 24957.828} C_VEL
LIN {X 0,Y 120.86,Z 986.819,A -85,B 0,C 180,E1 24958.962,E2 24958.962} C_VEL
LIN {X 0,Y 97.337,Z 990.257,A -85,B 0,C 180,E1 24974.787,E2 24974.787} C_VEL
LIN {X 0,Y 93.176,Z 1008.359,A -85,B 0,C 180,E1 24989.021,E2 24989.021} C_VEL
LIN {X 0,Y 93.539,Z 1020.045,A -85,B 0,C 180,E1 25002.577,E2 25002.577} C_VEL
LIN {X 0,Y 92.801,Z 1026.347,A -85,B 0,C 180,E1 25012.65,E2 25012.65} C_VEL
LIN {X 0,Y 95.128,Z 1031.334,A -85,B 0,C 180,E1 25022.821,E2 25022.821} C_VEL
LIN {X 0,Y 110.322,Z 1036.047,A -85,B 0,C 180,E1 25036.029,E2 25036.029} C_VEL
LIN {X 0,Y 131.84,Z 1036.132,A -85,B 0,C 180,E1 25046.403,E2 25046.403} C_VEL
LIN {X 0,Y 106.281,Z 1043.587,A -85,B 0,C 180,E1 25058.42,E2 25058.42} C_VEL
LIN {X 0,Y 88.203,Z 1046.297,A -85,B 0,C 180,E1 25079.008,E2 25079.008} C_VEL
LIN {X 0,Y 85.098,Z 1045.966,A -85,B 0,C 180,E1 25090.516,E2 25090.516} C_VEL
LIN {X 0,Y 84.799,Z 1052.551,A -85,B 0,C 180,E1 25110.004,E2 25110.004} C_VEL
LIN {X 0,Y 84.363,Z 1052.99,A -85,B 0,C 180,E1 25131.039,E2 25131.039} C_VEL
LIN {X 0,Y 93.359,Z 1048.776,A -85,B 0,C 180,E1 25150.449,E2 25150.449} C_VEL
LIN {X 0,Y 112.943,Z 1038.824,A -85,B 0,C 180,E1 25166.203,E2 25166.203} C_VEL
LIN {X 0,Y 138.407,Z 1022.691,A -85,B 0,C 180,E1 25176.378,E2 25176.378} C_VEL
LIN {X 0,Y 163.387,Z 1001.986,A -85,B 0,C 180,E1 25182.254,E2 25182.254} C_VEL
LIN {X 0,Y 165.329,Z 999.541,A -85,B 0,C 180,E1 25183.278,E2 25183.278} C_VEL
LIN {X 0,Y 166.347,Z 994.119,A -85,B 0,C 180,E1 25189.448,E2 25189.448} C_VEL
LIN {X 0,Y 166.768,Z 991.212,A -85,B 0,C 180,E1 25194.726,E2 25194.726} C_VEL
LIN {X 0,Y 164.672,Z 991.978,A -85,B 0,C 180,E1 25199.933,E2 25199.933} C_VEL
LIN {X 0,Y 159.169,Z 996.912,A -85,B 0,C 180,E1 25208.129,E2 25208.129} C_VEL
LIN {X 0,Y 152.176,Z 1003.522,A -85,B 0,C 180,E1 25214.712,E2 25214.712} C_VEL
LIN {X 0,Y 130.647,Z 1017.037,A -85,B 0,C 180,E1 25222.003,E2 25222.003} C_VEL
LIN {X 0,Y 109.149,Z 1026.233,A -85,B 0,C 180,E1 25233.659,E2 25233.659} C_VEL
LIN {X 0,Y 93.486,Z 1029.592,A -85,B 0,C 180,E1 25249.617,E2 25249.617} C_VEL
LIN {X 0,Y 86.014,Z 1027.65,A -85,B 0,C 180,E1 25269.383,E2 25269.383} C_VEL
LIN {X 0,Y 88.535,Z 1020.393,A -85,B 0,C 180,E1 25289.997,E2 25289.997} C_VEL
LIN {X 0,Y 99.374,Z 1007.41,A -85,B 0,C 180,E1 25307.738,E2 25307.738} C_VEL
LIN {X 0,Y 110.93,Z 994.068,A -85,B 0,C 180,E1 25317.678,E2 25317.678} C_VEL
LIN {X 0,Y 111.13,Z 992.624,A -85,B 0,C 180,E1 25319.183,E2 25319.183} C_VEL
LIN {X 0,Y 88.336,Z 995.836,A -85,B 0,C 180,E1 25336.913,E2 25336.913} C_VEL
LIN {X 0,Y 87.122,Z 998.923,A -85,B 0,C 180,E1 25340.319,E2 25340.319} C_VEL
LIN {X 0,Y 84.999,Z 1015.921,A -85,B 0,C 180,E1 25357.754,E2 25357.754} C_VEL
LIN {X 0,Y 90.971,Z 1028.431,A -85,B 0,C 180,E1 25376.922,E2 25376.922} C_VEL
LIN {X 0,Y 95.128,Z 1031.334,A -85,B 0,C 180,E1 25382.821,E2 25382.821} C_VEL
LIN {X 0,Y 100.319,Z 1035.183,A -85,B 0,C 180,E1 25392.382,E2 25392.382} C_VEL
LIN {X 0,Y 107.783,Z 1037.689,A -85,B 0,C 180,E1 25400.69,E2 25400.69} C_VEL
LIN {X 0,Y 108.157,Z 1037.555,A -85,B 0,C 180,E1 25400.899,E2 25400.899} C_VEL
LIN {X 0,Y 117.199,Z 1038.358,A -85,B 0,C 180,E1 25405.274,E2 25405.274} C_VEL
LIN {X 0,Y 118.728,Z 1038.642,A -85,B 0,C 180,E1 25406.794,E2 25406.794} C_VEL
LIN {X 0,Y 94.048,Z 1043.601,A -85,B 0,C 180,E1 25420.221,E2 25420.221} C_VEL
LIN {X 0,Y 78.305,Z 1043.625,A -85,B 0,C 180,E1 25446.02,E2 25446.02} C_VEL
LIN {X 0,Y 76.926,Z 1051.188,A -85,B 0,C 180,E1 25470.004,E2 25470.004} C_VEL
LIN {X 0,Y 76.877,Z 1051.793,A -85,B 0,C 180,E1 25493.201,E2 25493.201} C_VEL
LIN {X 0,Y 89.713,Z 1046.79,A -85,B 0,C 180,E1 25516.439,E2 25516.439} C_VEL
LIN {X 0,Y 112.542,Z 1035.949,A -85,B 0,C 180,E1 25531.585,E2 25531.585} C_VEL
LIN {X 0,Y 138.287,Z 1020.044,A -85,B 0,C 180,E1 25540.252,E2 25540.252} C_VEL
LIN {X 0,Y 158.442,Z 1004.021,A -85,B 0,C 180,E1 25544.518,E2 25544.518} C_VEL
LIN {X 0,Y 159.895,Z 1001.283,A -85,B 0,C 180,E1 25546.807,E2 25546.807} C_VEL
LIN {X 0,Y 160.74,Z 996.597,A -85,B 0,C 180,E1 25554.528,E2 25554.528} C_VEL
LIN {X 0,Y 158.438,Z 997.298,A -85,B 0,C 180,E1 25559.93,E2 25559.93} C_VEL
LIN {X 0,Y 152.736,Z 1001.624,A -85,B 0,C 180,E1 25567.546,E2 25567.546} C_VEL
LIN {X 0,Y 147.226,Z 1006.163,A -85,B 0,C 180,E1 25572.481,E2 25572.481} C_VEL
LIN {X 0,Y 125.143,Z 1019.026,A -85,B 0,C 180,E1 25579.587,E2 25579.587} C_VEL
LIN {X 0,Y 104.79,Z 1027.178,A -85,B 0,C 180,E1 25589.891,E2 25589.891} C_VEL
LIN {X 0,Y 87.38,Z 1030.74,A -85,B 0,C 180,E1 25606.119,E2 25606.119} C_VEL
LIN {X 0,Y 78.467,Z 1029.034,A -85,B 0,C 180,E1 25627.295,E2 25627.295} C_VEL
LIN {X 0,Y 80.479,Z 1022.049,A -85,B 0,C 180,E1 25649.996,E2 25649.996} C_VEL
LIN {X 0,Y 91.853,Z 1009.366,A -85,B 0,C 180,E1 25669.245,E2 25669.245} C_VEL
LIN {X 0,Y 102.089,Z 998.459,A -85,B 0,C 180,E1 25678.375,E2 25678.375} C_VEL
LIN {X 0,Y 78.642,Z 1001.44,A -85,B 0,C 180,E1 25702.142,E2 25702.142} C_VEL
LIN {X 0,Y 77.527,Z 1018.11,A -85,B 0,C 180,E1 25721.557,E2 25721.557} C_VEL
LIN {X 0,Y 86.227,Z 1030.661,A -85,B 0,C 180,E1 25742.646,E2 25742.646} C_VEL
LIN {X 0,Y 102.182,Z 1036.807,A -85,B 0,C 180,E1 25757.345,E2 25757.345} C_VEL
LIN {X 0,Y 108.157,Z 1037.555,A -85,B 0,C 180,E1 25760.899,E2 25760.899} C_VEL
LIN {X 0,Y 108.487,Z 1038.67,A -85,B 0,C 180,E1 25763.815,E2 25763.815} C_VEL
LIN {X 0,Y 103.476,Z 1040.093,A -85,B 0,C 180,E1 25767.577,E2 25767.577} C_VEL
LIN {X 0,Y 95.62,Z 1041.235,A -85,B 0,C 180,E1 25771.946,E2 25771.946} C_VEL
LIN {X 0,Y 75.086,Z 1042.316,A -85,B 0,C 180,E1 25792.781,E2 25792.781} C_VEL
LIN {X 0,Y 71.135,Z 1041.709,A -85,B 0,C 180,E1 25803.492,E2 25803.492} C_VEL
LIN {X 0,Y 68.522,Z 1048.179,A -85,B 0,C 180,E1 25822.47,E2 25822.47} C_VEL
LIN {X 0,Y 69.057,Z 1049.819,A -85,B 0,C 180,E1 25830.004,E2 25830.004} C_VEL
LIN {X 0,Y 69.535,Z 1050.598,A -85,B 0,C 180,E1 25855.821,E2 25855.821} C_VEL
LIN {X 0,Y 81.705,Z 1046.66,A -85,B 0,C 180,E1 25877.843,E2 25877.843} C_VEL
LIN {X 0,Y 105.379,Z 1036.832,A -85,B 0,C 180,E1 25893.828,E2 25893.828} C_VEL
LIN {X 0,Y 130.645,Z 1022.826,A -85,B 0,C 180,E1 25902.227,E2 25902.227} C_VEL
LIN {X 0,Y 152.924,Z 1006.606,A -85,B 0,C 180,E1 25906.77,E2 25906.77} C_VEL
LIN {X 0,Y 154.073,Z 1003.355,A -85,B 0,C 180,E1 25911.081,E2 25911.081} C_VEL
LIN {X 0,Y 154.477,Z 1001.746,A -85,B 0,C 180,E1 25914.305,E2 25914.305} C_VEL
LIN {X 0,Y 151.422,Z 1002.656,A -85,B 0,C 180,E1 25920.62,E2 25920.62} C_VEL
LIN {X 0,Y 145.021,Z 1006.933,A -85,B 0,C 180,E1 25927.95,E2 25927.95} C_VEL
LIN {X 0,Y 142.178,Z 1008.961,A -85,B 0,C 180,E1 25930.157,E2 25930.157} C_VEL
LIN {X 0,Y 118.952,Z 1021.444,A -85,B 0,C 180,E1 25937.316,E2 25937.316} C_VEL
LIN {X 0,Y 98.432,Z 1028.813,A -85,B 0,C 180,E1 25947.341,E2 25947.341} C_VEL
LIN {X 0,Y 81.649,Z 1031.889,A -85,B 0,C 180,E1 25962.114,E2 25962.114} C_VEL
LIN {X 0,Y 71.018,Z 1030.414,A -85,B 0,C 180,E1 25984.756,E2 25984.756} C_VEL
LIN {X 0,Y 72.397,Z 1023.693,A -85,B 0,C 180,E1 26009.996,E2 26009.996} C_VEL
LIN {X 0,Y 84.415,Z 1011.302,A -85,B 0,C 180,E1 26031.018,E2 26031.018} C_VEL
LIN {X 0,Y 92.096,Z 1003.814,A -85,B 0,C 180,E1 26038.203,E2 26038.203} C_VEL
LIN {X 0,Y 91.073,Z 1003.263,A -85,B 0,C 180,E1 26039.913,E2 26039.913} C_VEL
LIN {X 0,Y 69.673,Z 1006.471,A -85,B 0,C 180,E1 26067.342,E2 26067.342} C_VEL
LIN {X 0,Y 71.694,Z 1023.185,A -85,B 0,C 180,E1 26091.05,E2 26091.05} C_VEL
LIN {X 0,Y 83.894,Z 1033.595,A -85,B 0,C 180,E1 26110.527,E2 26110.527} C_VEL
LIN {X 0,Y 105.936,Z 1039.325,A -85,B 0,C 180,E1 26125.494,E2 26125.494} C_VEL
LIN {X 0,Y 102.929,Z 1040.261,A -85,B 0,C 180,E1 26128.049,E2 26128.049} C_VEL
LIN {X 0,Y 95.62,Z 1041.235,A -85,B 0,C 180,E1 26131.946,E2 26131.946} C_VEL
LIN {X 0,Y 81.517,Z 1041.545,A -85,B 0,C 180,E1 26138.679,E2 26138.679} C_VEL
LIN {X 0,Y 69.348,Z 1040.138,A -85,B 0,C 180,E1 26148.222,E2 26148.222} C_VEL
LIN {X 0,Y 64.421,Z 1039.785,A -85,B 0,C 180,E1 26159.485,E2 26159.485} C_VEL
LIN {X 0,Y 60.84,Z 1047.844,A -85,B 0,C 180,E1 26186.564,E2 26186.564} C_VEL
LIN {X 0,Y 60.772,Z 1048.698,A -85,B 0,C 180,E1 26192.11,E2 26192.11} C_VEL
LIN {X 0,Y 62.37,Z 1049.372,A -85,B 0,C 180,E1 26219.052,E2 26219.052} C_VEL
LIN {X 0,Y 79.435,Z 1044.681,A -85,B 0,C 180,E1 26244.97,E2 26244.97} C_VEL
LIN {X 0,Y 105.202,Z 1034.525,A -85,B 0,C 180,E1 26259.129,E2 26259.129} C_VEL
LIN {X 0,Y 133.283,Z 1019.067,A -85,B 0,C 180,E1 26266.664,E2 26266.664} C_VEL
LIN {X 0,Y 145.325,Z 1010.727,A -85,B 0,C 180,E1 26268.823,E2 26268.823} C_VEL
LIN {X 0,Y 147.477,Z 1008.736,A -85,B 0,C 180,E1 26269.834,E2 26269.834} C_VEL
LIN {X 0,Y 148.005,Z 1006.632,A -85,B 0,C 180,E1 26274.056,E2 26274.056} C_VEL
LIN {X 0,Y 145.186,Z 1007.209,A -85,B 0,C 180,E1 26279.924,E2 26279.924} C_VEL
LIN {X 0,Y 139.43,Z 1010.438,A -85,B 0,C 180,E1 26286.151,E2 26286.151} C_VEL
LIN {X 0,Y 137.495,Z 1011.583,A -85,B 0,C 180,E1 26287.648,E2 26287.648} C_VEL
LIN {X 0,Y 113.444,Z 1023.591,A -85,B 0,C 180,E1 26294.609,E2 26294.609} C_VEL
LIN {X 0,Y 90.045,Z 1030.952,A -85,B 0,C 180,E1 26305.889,E2 26305.889} C_VEL
LIN {X 0,Y 76.386,Z 1033.037,A -85,B 0,C 180,E1 26317.54,E2 26317.54} C_VEL
LIN {X 0,Y 63.764,Z 1031.794,A -85,B 0,C 180,E1 26341.641,E2 26341.641} C_VEL
LIN {X 0,Y 64.334,Z 1025.311,A -85,B 0,C 180,E1 26369.995,E2 26369.995} C_VEL
LIN {X 0,Y 77.074,Z 1013.19,A -85,B 0,C 180,E1 26393.13,E2 26393.13} C_VEL
LIN {X 0,Y 82.71,Z 1008.086,A -85,B 0,C 180,E1 26398.698,E2 26398.698} C_VEL
LIN {X 0,Y 61.241,Z 1011.503,A -85,B 0,C 180,E1 26434.576,E2 26434.576} C_VEL
LIN {X 0,Y 67.234,Z 1026.834,A -85,B 0,C 180,E1 26460.165,E2 26460.165} C_VEL
LIN {X 0,Y 81.995,Z 1035.847,A -85,B 0,C 180,E1 26477.73,E2 26477.73} C_VEL
LIN {X 0,Y 94.365,Z 1039.374,A -85,B 0,C 180,E1 26485.682,E2 26485.682} C_VEL
LIN {X 0,Y 77.103,Z 1040.588,A -85,B 0,C 180,E1 26498.241,E2 26498.241} C_VEL
LIN {X 0,Y 69.348,Z 1040.138,A -85,B 0,C 180,E1 26508.222,E2 26508.222} C_VEL
LIN {X 0,Y 62.102,Z 1040.714,A -85,B 0,C 180,E1 26517.74,E2 26517.74} C_VEL
LIN {X 0,Y 53.078,Z 1044.238,A -85,B 0,C 180,E1 26535.199,E2 26535.199} C_VEL
LIN {X 0,Y 52.868,Z 1044.694,A -85,B 0,C 180,E1 26537.518,E2 26537.518} C_VEL
LIN {X 0,Y 53.275,Z 1047.08,A -85,B 0,C 180,E1 26550.006,E2 26550.006} C_VEL
LIN {X 0,Y 55.449,Z 1048.124,A -85,B 0,C 180,E1 26583.108,E2 26583.108} C_VEL
LIN {X 0,Y 75.064,Z 1043.631,A -85,B 0,C 180,E1 26610.059,E2 26610.059} C_VEL
LIN {X 0,Y 102.917,Z 1033.543,A -85,B 0,C 180,E1 26623.455,E2 26623.455} C_VEL
LIN {X 0,Y 131.655,Z 1018.438,A -85,B 0,C 180,E1 26630.085,E2 26630.085} C_VEL
LIN {X 0,Y 139.953,Z 1012.996,A -85,B 0,C 180,E1 26631.394,E2 26631.394} C_VEL
LIN {X 0,Y 141.343,Z 1011.246,A -85,B 0,C 180,E1 26633.774,E2 26633.774} C_VEL
LIN {X 0,Y 138.066,Z 1011.848,A -85,B 0,C 180,E1 26639.92,E2 26639.92} C_VEL
LIN {X 0,Y 133.555,Z 1013.991,A -85,B 0,C 180,E1 26644.49,E2 26644.49} C_VEL
LIN {X 0,Y 108.211,Z 1025.656,A -85,B 0,C 180,E1 26651.625,E2 26651.625} C_VEL
LIN {X 0,Y 82.585,Z 1032.749,A -85,B 0,C 180,E1 26663.545,E2 26663.545} C_VEL
LIN {X 0,Y 62.769,Z 1034.326,A -85,B 0,C 180,E1 26683.637,E2 26683.637} C_VEL
LIN {X 0,Y 54.418,Z 1030.691,A -85,B 0,C 180,E1 26713.839,E2 26713.839} C_VEL
LIN {X 0,Y 62.695,Z 1020.954,A -85,B 0,C 180,E1 26745.745,E2 26745.745} C_VEL
LIN {X 0,Y 73.03,Z 1012.356,A -85,B 0,C 180,E1 26759.099,E2 26759.099} C_VEL
LIN {X 0,Y 54.034,Z 1016.15,A -85,B 0,C 180,E1 26803.948,E2 26803.948} C_VEL
LIN {X 0,Y 65.327,Z 1030.705,A -85,B 0,C 180,E1 26831.158,E2 26831.158} C_VEL
LIN {X 0,Y 82.212,Z 1038.308,A -85,B 0,C 180,E1 26845.65,E2 26845.65} C_VEL
LIN {X 0,Y 58.845,Z 1037.141,A -85,B 0,C 180,E1 26873.065,E2 26873.065} C_VEL
LIN {X 0,Y 52.868,Z 1044.694,A -85,B 0,C 180,E1 26897.518,E2 26897.518} C_VEL
LIN {X 0,Y 50.432,Z 1046.504,A -85,B 0,C 180,E1 26909.042,E2 26909.042} C_VEL
LIN {X 0,Y 46.074,Z 1046.908,A -85,B 0,C 180,E1 26938.659,E2 26938.659} C_VEL
LIN {X 0,Y 62.136,Z 1044.754,A -85,B 0,C 180,E1 26968.532,E2 26968.532} C_VEL
LIN {X 0,Y 90.295,Z 1036.83,A -85,B 0,C 180,E1 26984.629,E2 26984.629} C_VEL
LIN {X 0,Y 122.235,Z 1022.581,A -85,B 0,C 180,E1 26992.294,E2 26992.294} C_VEL
LIN {X 0,Y 134.005,Z 1015.556,A -85,B 0,C 180,E1 26994.434,E2 26994.434} C_VEL
LIN {X 0,Y 130.704,Z 1016.197,A -85,B 0,C 180,E1 26999.915,E2 26999.915} C_VEL
LIN {X 0,Y 127.338,Z 1017.627,A -85,B 0,C 180,E1 27002.354,E2 27002.354} C_VEL
LIN {X 0,Y 98.039,Z 1029.397,A -85,B 0,C 180,E1 27009.993,E2 27009.993} C_VEL
LIN {X 0,Y 79.651,Z 1033.789,A -85,B 0,C 180,E1 27018.101,E2 27018.101} C_VEL
LIN {X 0,Y 57.419,Z 1035.575,A -85,B 0,C 180,E1 27037.706,E2 27037.706} C_VEL
LIN {X 0,Y 46.677,Z 1032.13,A -85,B 0,C 180,E1 27071.065,E2 27071.065} C_VEL
LIN {X 0,Y 54.08,Z 1023.361,A -85,B 0,C 180,E1 27106.253,E2 27106.253} C_VEL
LIN {X 0,Y 62.786,Z 1016.858,A -85,B 0,C 180,E1 27118.83,E2 27118.83} C_VEL
LIN {X 0,Y 48.754,Z 1020.847,A -85,B 0,C 180,E1 27176.683,E2 27176.683} C_VEL
LIN {X 0,Y 65.23,Z 1033.98,A -85,B 0,C 180,E1 27201.817,E2 27201.817} C_VEL
LIN {X 0,Y 70.24,Z 1036.204,A -85,B 0,C 180,E1 27205.702,E2 27205.702} C_VEL
LIN {X 0,Y 53.624,Z 1034.825,A -85,B 0,C 180,E1 27226.344,E2 27226.344} C_VEL
LIN {X 0,Y 45.014,Z 1044.204,A -85,B 0,C 180,E1 27260.325,E2 27260.325} C_VEL
LIN {X 0,Y 45.357,Z 1045.708,A -85,B 0,C 180,E1 27270.007,E2 27270.007} C_VEL
LIN {X 0,Y 46.074,Z 1046.908,A -85,B 0,C 180,E1 27298.659,E2 27298.659} C_VEL
LIN {X 0,Y 47.817,Z 1046.677,A -85,B 0,C 180,E1 27309.102,E2 27309.102} C_VEL
LIN {X 0,Y 56.674,Z 1043.984,A -85,B 0,C 180,E1 27333.863,E2 27333.863} C_VEL
LIN {X 0,Y 58.278,Z 1043.649,A -85,B 0,C 180,E1 27335.31,E2 27335.31} C_VEL
LIN {X 0,Y 90.593,Z 1035.184,A -85,B 0,C 180,E1 27350.259,E2 27350.259} C_VEL
LIN {X 0,Y 121.42,Z 1021.916,A -85,B 0,C 180,E1 27356.051,E2 27356.051} C_VEL
LIN {X 0,Y 125.233,Z 1019.698,A -85,B 0,C 180,E1 27357.071,E2 27357.071} C_VEL
LIN {X 0,Y 121.133,Z 1021.233,A -85,B 0,C 180,E1 27359.758,E2 27359.758} C_VEL
LIN {X 0,Y 91.502,Z 1031.815,A -85,B 0,C 180,E1 27366.846,E2 27366.846} C_VEL
LIN {X 0,Y 64.39,Z 1036.476,A -85,B 0,C 180,E1 27379.838,E2 27379.838} C_VEL
LIN {X 0,Y 43.775,Z 1035.823,A -85,B 0,C 180,E1 27406.221,E2 27406.221} C_VEL
LIN {X 0,Y 40.089,Z 1030.016,A -85,B 0,C 180,E1 27449.992,E2 27449.992} C_VEL
LIN {X 0,Y 50.844,Z 1022.099,A -85,B 0,C 180,E1 27476.433,E2 27476.433} C_VEL
LIN {X 0,Y 52.48,Z 1020.628,A -85,B 0,C 180,E1 27480.521,E2 27480.521} C_VEL
LIN {X 0,Y 46.346,Z 1025.162,A -85,B 0,C 180,E1 27551.491,E2 27551.491} C_VEL
LIN {X 0,Y 58.774,Z 1033.229,A -85,B 0,C 180,E1 27566.236,E2 27566.236} C_VEL
LIN {X 0,Y 49.988,Z 1032.048,A -85,B 0,C 180,E1 27577.545,E2 27577.545} C_VEL
LIN {X 0,Y 37.216,Z 1042.756,A -85,B 0,C 180,E1 27618.271,E2 27618.271} C_VEL
LIN {X 0,Y 37.454,Z 1044.324,A -85,B 0,C 180,E1 27630.008,E2 27630.008} C_VEL
LIN {X 0,Y 42.87,Z 1045.631,A -85,B 0,C 180,E1 27674.949,E2 27674.949} C_VEL
LIN {X 0,Y 58.278,Z 1043.649,A -85,B 0,C 180,E1 27695.31,E2 27695.31} C_VEL
LIN {X 0,Y 70.18,Z 1040.401,A -85,B 0,C 180,E1 27706.493,E2 27706.493} C_VEL
LIN {X 0,Y 83.773,Z 1036.076,A -85,B 0,C 180,E1 27714.088,E2 27714.088} C_VEL
LIN {X 0,Y 106.032,Z 1028.145,A -85,B 0,C 180,E1 27718.399,E2 27718.399} C_VEL
LIN {X 0,Y 76.156,Z 1035.856,A -85,B 0,C 180,E1 27726.207,E2 27726.207} C_VEL
LIN {X 0,Y 49.13,Z 1037.993,A -85,B 0,C 180,E1 27742.384,E2 27742.384} C_VEL
LIN {X 0,Y 31.733,Z 1035.009,A -85,B 0,C 180,E1 27781.491,E2 27781.491} C_VEL
LIN {X 0,Y 38.873,Z 1026.768,A -85,B 0,C 180,E1 27832.914,E2 27832.914} C_VEL
LIN {X 0,Y 42.809,Z 1024.47,A -85,B 0,C 180,E1 27839.617,E2 27839.617} C_VEL
LIN {X 0,Y 47.537,Z 1029.442,A -85,B 0,C 180,E1 27927.73,E2 27927.73} C_VEL
LIN {X 0,Y 29.484,Z 1041.31,A -85,B 0,C 180,E1 27975.132,E2 27975.132} C_VEL
LIN {X 0,Y 29.526,Z 1042.932,A -85,B 0,C 180,E1 27990.01,E2 27990.01} C_VEL
LIN {X 0,Y 37.583,Z 1044.383,A -85,B 0,C 180,E1 28043.694,E2 28043.694} C_VEL
LIN {X 0,Y 62.231,Z 1041.32,A -85,B 0,C 180,E1 28066.727,E2 28066.727} C_VEL
LIN {X 0,Y 83.773,Z 1036.076,A -85,B 0,C 180,E1 28074.088,E2 28074.088} C_VEL
LIN {X 0,Y 82.158,Z 1036.001,A -85,B 0,C 180,E1 28076.614,E2 28076.614} C_VEL
LIN {X 0,Y 71.501,Z 1037.535,A -85,B 0,C 180,E1 28080.947,E2 28080.947} C_VEL
LIN {X 0,Y 63.825,Z 1038.302,A -85,B 0,C 180,E1 28083.837,E2 28083.837} C_VEL
LIN {X 0,Y 34.768,Z 1038.57,A -85,B 0,C 180,E1 28105.45,E2 28105.45} C_VEL
LIN {X 0,Y 23.913,Z 1033.129,A -85,B 0,C 180,E1 28169.987,E2 28169.987} C_VEL
LIN {X 0,Y 31.594,Z 1028.441,A -85,B 0,C 180,E1 28198.624,E2 28198.624} C_VEL
LIN {X 0,Y 32.199,Z 1027.814,A -85,B 0,C 180,E1 28202.902,E2 28202.902} C_VEL
LIN {X 0,Y 35.519,Z 1031.71,A -85,B 0,C 180,E1 28285.565,E2 28285.565} C_VEL
LIN {X 0,Y 21.868,Z 1039.836,A -85,B 0,C 180,E1 28329.761,E2 28329.761} C_VEL
LIN {X 0,Y 21.604,Z 1041.495,A -85,B 0,C 180,E1 28350.014,E2 28350.014} C_VEL
LIN {X 0,Y 33.44,Z 1043.137,A -85,B 0,C 180,E1 28414.919,E2 28414.919} C_VEL
LIN {X 0,Y 60.884,Z 1040.231,A -85,B 0,C 180,E1 28434.164,E2 28434.164} C_VEL
LIN {X 0,Y 79.163,Z 1036.234,A -85,B 0,C 180,E1 28439.075,E2 28439.075} C_VEL
LIN {X 0,Y 63.825,Z 1038.302,A -85,B 0,C 180,E1 28443.837,E2 28443.837} C_VEL
LIN {X 0,Y 55.39,Z 1039.562,A -85,B 0,C 180,E1 28443.669,E2 28443.669} C_VEL
LIN {X 0,Y 41.492,Z 1041.281,A -85,B 0,C 180,E1 28435.671,E2 28435.671} C_VEL
LIN {X 0,Y 18.209,Z 1041.553,A -85,B 0,C 180,E1 28406.282,E2 28406.282} C_VEL
LIN {X 0,Y 13.672,Z 1040.048,A -85,B 0,C 180,E1 28350.022,E2 28350.022} C_VEL
LIN {X 0,Y 20.891,Z 1035.262,A -85,B 0,C 180,E1 28290.368,E2 28290.368} C_VEL
LIN {X 0,Y 23.248,Z 1033.695,A -85,B 0,C 180,E1 28280.407,E2 28280.407} C_VEL
LIN {X 0,Y 22.631,Z 1030.978,A -85,B 0,C 180,E1 28203.238,E2 28203.238} C_VEL
LIN {X 0,Y 19.089,Z 1037.876,A -85,B 0,C 180,E1 28117.49,E2 28117.49} C_VEL
LIN {X 0,Y 45.485,Z 1040.416,A -85,B 0,C 180,E1 28082.885,E2 28082.885} C_VEL
LIN {X 0,Y 52.494,Z 1040.295,A -85,B 0,C 180,E1 28079.789,E2 28079.789} C_VEL
LIN {X 0,Y 41.492,Z 1041.281,A -85,B 0,C 180,E1 28075.671,E2 28075.671} C_VEL
LIN {X 0,Y 32.951,Z 1041.607,A -85,B 0,C 180,E1 28072.713,E2 28072.713} C_VEL
LIN {X 0,Y 8.415,Z 1039.533,A -85,B 0,C 180,E1 28051.767,E2 28051.767} C_VEL
LIN {X 0,Y 7.616,Z 1039.274,A -85,B 0,C 180,E1 28046.365,E2 28046.365} C_VEL
LIN {X 0,Y 5.756,Z 1038.608,A -85,B 0,C 180,E1 27990.053,E2 27990.053} C_VEL
LIN {X 0,Y 9.433,Z 1036.608,A -85,B 0,C 180,E1 27928.142,E2 27928.142} C_VEL
LIN {X 0,Y 12.053,Z 1035.372,A -85,B 0,C 180,E1 27911.104,E2 27911.104} C_VEL
LIN {X 0,Y 11.452,Z 1034.373,A -85,B 0,C 180,E1 27844.618,E2 27844.618} C_VEL
LIN {X 0,Y 15.536,Z 1039.266,A -85,B 0,C 180,E1 27732.857,E2 27732.857} C_VEL
LIN {X 0,Y 22.148,Z 1040.545,A -85,B 0,C 180,E1 27719.499,E2 27719.499} C_VEL
LIN {X 0,Y 7.616,Z 1039.274,A -85,B 0,C 180,E1 27686.365,E2 27686.365} C_VEL
LIN {X 0,Y 6.331,Z 1041.264,A -85,B 0,C 180,E1 27671.552,E2 27671.552} C_VEL
LIN {X 0,Y 6.331,Z 1116.5,A -85,B 0,C 180,E1 27671.552,E2 27671.552} C_VEL
LIN {X 0,Y 6.331,Z 1116.5,A -85,B 0,C 180,E1 27671.552,E2 27671.552}

QRS_NEXT_CUT()
PTP {E1 27537.074,E2 27537.074}
PTP {X 0,Y 607.913,A -85,B 0,C 180,E1 27537.074,E2 27537.074,E3 0,E4 0,E5 0,E6 0}
QRS_SPEED_INIT()
LIN {X 0,Y 607.913,Z 1116.5,A -85,B 0,C 180,E1 27537.074,E2 27537.074,E3 0,E4 0,E5 0,E6 0} C_VEL
LIN {X 0,Y 607.913,Z 674.985,A -85,B 0,C 180,E1 27537.074,E2 27537.074} C_VEL
LIN {X 0,Y 607.913,Z 665.752,A -85,B 0,C 180,E1 27537.074,E2 27537.074} C_VEL
LIN {X 0,Y 607.889,Z 664.253,A -85,B 0,C 180,E1 27536.761,E2 27536.761} C_VEL
LIN {X 0,Y 607.916,Z 692.729,A -85,B 0,C 180,E1 27533.768,E2 27533.768} C_VEL
LIN {X 0,Y 607.919,Z 832.471,A -85,B 0,C 180,E1 27532.059,E2 27532.059} C_VEL
LIN {X 0,Y 607.919,Z 848.94,A -85,B 0,C 180,E1 27531.678,E2 27531.678} C_VEL
LIN {X 0,Y 607.912,Z 864.172,A -85,B 0,C 180,E1 27531.154,E2 27531.154} C_VEL
LIN {X 0,Y 607.913,Z 879.321,A -85,B 0,C 180,E1 27530.438,E2 27530.438} C_VEL
LIN {X 0,Y 607.92,Z 893.472,A -85,B 0,C 180,E1 27529.576,E2 27529.576} C_VEL
LIN {X 0,Y 607.918,Z 906.188,A -85,B 0,C 180,E1 27528.598,E2 27528.598} C_VEL
LIN {X 0,Y 607.919,Z 918.108,A -85,B 0,C 180,E1 27527.461,E2 27527.461} C_VEL
LIN {X 0,Y 607.919,Z 928.623,A -85,B 0,C 180,E1 27526.203,E2 27526.203} C_VEL
LIN {X 0,Y 607.916,Z 937.666,A -85,B 0,C 180,E1 27524.84,E2 27524.84} C_VEL
LIN {X 0,Y 607.917,Z 944.685,A -85,B 0,C 180,E1 27523.469,E2 27523.469} C_VEL
LIN {X 0,Y 607.913,Z 950.457,A -85,B 0,C 180,E1 27521.928,E2 27521.928} C_VEL
LIN {X 0,Y 607.914,Z 954.125,A -85,B 0,C 180,E1 27520.465,E2 27520.465} C_VEL
LIN {X 0,Y 607.914,Z 956.142,A -85,B 0,C 180,E1 27518.887,E2 27518.887} C_VEL
LIN {X 0,Y 607.916,Z 956.35,A -85,B 0,C 180,E1 27517.324,E2 27517.324} C_VEL
LIN {X 0,Y 607.915,Z 954.589,A -85,B 0,C 180,E1 27515.721,E2 27515.721} C_VEL
LIN {X 0,Y 607.915,Z 951.019,A -85,B 0,C 180,E1 27514.16,E2 27514.16} C_VEL
LIN {X 0,Y 607.914,Z 945.548,A -85,B 0,C 180,E1 27512.643,E2 27512.643} C_VEL
LIN {X 0,Y 607.914,Z 938.363,A -85,B 0,C 180,E1 27511.19,E2 27511.19} C_VEL
LIN {X 0,Y 607.917,Z 929.981,A -85,B 0,C 180,E1 27509.891,E2 27509.891} C_VEL
LIN {X 0,Y 607.919,Z 919.269,A -85,B 0,C 180,E1 27508.575,E2 27508.575} C_VEL
LIN {X 0,Y 607.917,Z 907.933,A -85,B 0,C 180,E1 27507.464,E2 27507.464} C_VEL
LIN {X 0,Y 607.919,Z 894.374,A -85,B 0,C 180,E1 27506.396,E2 27506.396} C_VEL
LIN {X 0,Y 607.909,Z 880.611,A -85,B 0,C 180,E1 27505.542,E2 27505.542} C_VEL
LIN {X 0,Y 607.909,Z 865.898,A -85,B 0,C 180,E1 27504.83,E2 27504.83} C_VEL
LIN {X 0,Y 607.918,Z 850.503,A -85,B 0,C 180,E1 27504.276,E2 27504.276} C_VEL
LIN {X 0,Y 607.918,Z 834.69,A -85,B 0,C 180,E1 27503.893,E2 27503.893} C_VEL
LIN {X 0,Y 607.895,Z 808.719,A -85,B 0,C 180,E1 27503.543,E2 27503.543} C_VEL
LIN {X 0,Y 607.904,Z 692.573,A -85,B 0,C 180,E1 27502.132,E2 27502.132} C_VEL
LIN {X 0,Y 607.891,Z 663.869,A -85,B 0,C 180,E1 27499.108,E2 27499.108} C_VEL
LIN {X 0,Y 607.917,Z 635.488,A -85,B 0,C 180,E1 27496.046,E2 27496.046} C_VEL
LIN {X 0,Y 607.917,Z 605.459,A -85,B 0,C 180,E1 27492.732,E2 27492.732} C_VEL
LIN {X 0,Y 607.916,Z 598.62,A -85,B 0,C 180,E1 27491.936,E2 27491.936} C_VEL
LIN {X 0,Y 607.839,Z 598.513,A -85,B 0,C 180,E1 27488.917,E2 27488.917} C_VEL
LIN {X 0,Y 607.882,Z 598.513,A -85,B 0,C 180,E1 27486.076,E2 27486.076} C_VEL
LIN {X 0,Y 607.852,Z 598.511,A -85,B 0,C 180,E1 27482.876,E2 27482.876} C_VEL
LIN {X 0,Y 607.868,Z 598.514,A -85,B 0,C 180,E1 27480.003,E2 27480.003} C_VEL
LIN {X 0,Y 607.86,Z 598.51,A -85,B 0,C 180,E1 27476.683,E2 27476.683} C_VEL
LIN {X 0,Y 607.872,Z 598.513,A -85,B 0,C 180,E1 27473.765,E2 27473.765} C_VEL
LIN {X 0,Y 607.87,Z 598.509,A -85,B 0,C 180,E1 27470.509,E2 27470.509} C_VEL
LIN {X 0,Y 607.868,Z 598.513,A -85,B 0,C 180,E1 27467.617,E2 27467.617} C_VEL
LIN {X 0,Y 607.877,Z 598.509,A -85,B 0,C 180,E1 27464.284,E2 27464.284} C_VEL
LIN {X 0,Y 607.879,Z 598.514,A -85,B 0,C 180,E1 27461.288,E2 27461.288} C_VEL
LIN {X 0,Y 607.907,Z 598.771,A -85,B 0,C 180,E1 27458.942,E2 27458.942} C_VEL
LIN {X 0,Y 607.915,Z 625.586,A -85,B 0,C 180,E1 27455.948,E2 27455.948} C_VEL
LIN {X 0,Y 607.885,Z 653.419,A -85,B 0,C 180,E1 27452.923,E2 27452.923} C_VEL
LIN {X 0,Y 607.917,Z 683.48,A -85,B 0,C 180,E1 27449.718,E2 27449.718} C_VEL
LIN {X 0,Y 607.888,Z 692.879,A -85,B 0,C 180,E1 27448.763,E2 27448.763} C_VEL
LIN {X 0,Y 607.917,Z 832.711,A -85,B 0,C 180,E1 27447.054,E2 27447.054} C_VEL
LIN {X 0,Y 607.919,Z 848.984,A -85,B 0,C 180,E1 27446.677,E2 27446.677} C_VEL
LIN {X 0,Y 607.915,Z 864.645,A -85,B 0,C 180,E1 27446.134,E2 27446.134} C_VEL
LIN {X 0,Y 607.913,Z 879.552,A -85,B 0,C 180,E1 27445.425,E2 27445.425} C_VEL
LIN {X 0,Y 607.919,Z 893.513,A -85,B 0,C 180,E1 27444.574,E2 27444.574} C_VEL
LIN {X 0,Y 607.918,Z 906.403,A -85,B 0,C 180,E1 27443.579,E2 27443.579} C_VEL
LIN {X 0,Y 607.918,Z 918.313,A -85,B 0,C 180,E1 27442.439,E2 27442.439} C_VEL
LIN {X 0,Y 607.917,Z 928.628,A -85,B 0,C 180,E1 27441.202,E2 27441.202} C_VEL
LIN {X 0,Y 607.916,Z 937.518,A -85,B 0,C 180,E1 27439.864,E2 27439.864} C_VEL
LIN {X 0,Y 607.916,Z 944.459,A -85,B 0,C 180,E1 27438.521,E2 27438.521} C_VEL
LIN {X 0,Y 607.916,Z 949.988,A -85,B 0,C 180,E1 27437.075,E2 27437.075} C_VEL
LIN {X 0,Y 607.919,Z 954.01,A -85,B 0,C 180,E1 27435.523,E2 27435.523} C_VEL
LIN {X 0,Y 607.914,Z 956.091,A -85,B 0,C 180,E1 27433.96,E2 27433.96} C_VEL
LIN {X 0,Y 607.916,Z 956.372,A -85,B 0,C 180,E1 27432.385,E2 27432.385} C_VEL
LIN {X 0,Y 607.918,Z 954.879,A -85,B 0,C 180,E1 27430.895,E2 27430.895} C_VEL
LIN {X 0,Y 607.918,Z 951.382,A -85,B 0,C 180,E1 27429.292,E2 27429.292} C_VEL
LIN {X 0,Y 607.918,Z 946.291,A -85,B 0,C 180,E1 27427.818,E2 27427.818} C_VEL
LIN {X 0,Y 607.918,Z 939.179,A -85,B 0,C 180,E1 27426.34,E2 27426.34} C_VEL
LIN {X 0,Y 607.918,Z 930.726,A -85,B 0,C 180,E1 27424.992,E2 27424.992} C_VEL
LIN {X 0,Y 607.918,Z 920.256,A -85,B 0,C 180,E1 27423.687,E2 27423.687} C_VEL
LIN {X 0,Y 607.918,Z 909.258,A -85,B 0,C 180,E1 27422.579,E2 27422.579} C_VEL
LIN {X 0,Y 607.919,Z 895.983,A -85,B 0,C 180,E1 27421.513,E2 27421.513} C_VEL
LIN {X 0,Y 607.918,Z 882.603,A -85,B 0,C 180,E1 27420.651,E2 27420.651} C_VEL
LIN {X 0,Y 607.907,Z 867.504,A -85,B 0,C 180,E1 27419.899,E2 27419.899} C_VEL
LIN {X 0,Y 607.919,Z 851.713,A -85,B 0,C 180,E1 27419.313,E2 27419.313} C_VEL
LIN {X 0,Y 607.917,Z 836.269,A -85,B 0,C 180,E1 27418.922,E2 27418.922} C_VEL
LIN {X 0,Y 607.916,Z 814.061,A -85,B 0,C 180,E1 27418.608,E2 27418.608} C_VEL
LIN {X 0,Y 607.896,Z 692.527,A -85,B 0,C 180,E1 27417.127,E2 27417.127} C_VEL
LIN {X 0,Y 607.913,Z 662.171,A -85,B 0,C 180,E1 27413.927,E2 27413.927} C_VEL
LIN {X 0,Y 607.896,Z 633.535,A -85,B 0,C 180,E1 27410.832,E2 27410.832} C_VEL
LIN {X 0,Y 607.919,Z 603.689,A -85,B 0,C 180,E1 27407.534,E2 27407.534} C_VEL
LIN {X 0,Y 607.911,Z 598.623,A -85,B 0,C 180,E1 27406.933,E2 27406.933} C_VEL
LIN {X 0,Y 607.9,Z 598.506,A -85,B 0,C 180,E1 27403.694,E2 27403.694} C_VEL
LIN {X 0,Y 607.901,Z 598.512,A -85,B 0,C 180,E1 27400.518,E2 27400.518} C_VEL
LIN {X 0,Y 607.898,Z 598.506,A -85,B 0,C 180,E1 27397.368,E2 27397.368} C_VEL
LIN {X 0,Y 607.899,Z 598.511,A -85,B 0,C 180,E1 27394.23,E2 27394.23} C_VEL
LIN {X 0,Y 607.9,Z 598.506,A -85,B 0,C 180,E1 27391.095,E2 27391.095} C_VEL
LIN {X 0,Y 607.897,Z 598.511,A -85,B 0,C 180,E1 27387.954,E2 27387.954} C_VEL
LIN {X 0,Y 607.899,Z 598.506,A -85,B 0,C 180,E1 27384.781,E2 27384.781} C_VEL
LIN {X 0,Y 607.894,Z 598.51,A -85,B 0,C 180,E1 27381.619,E2 27381.619} C_VEL
LIN {X 0,Y 607.9,Z 598.506,A -85,B 0,C 180,E1 27378.509,E2 27378.509} C_VEL
LIN {X 0,Y 607.892,Z 598.51,A -85,B 0,C 180,E1 27375.356,E2 27375.356} C_VEL
LIN {X 0,Y 607.901,Z 598.506,A -85,B 0,C 180,E1 27372.25,E2 27372.25} C_VEL
LIN {X 0,Y 607.891,Z 598.51,A -85,B 0,C 180,E1 27369.085,E2 27369.085} C_VEL
LIN {X 0,Y 607.901,Z 598.507,A -85,B 0,C 180,E1 27365.948,E2 27365.948} C_VEL
LIN {X 0,Y 607.89,Z 598.51,A -85,B 0,C 180,E1 27362.829,E2 27362.829} C_VEL
LIN {X 0,Y 607.903,Z 598.506,A -85,B 0,C 180,E1 27359.717,E2 27359.717} C_VEL
LIN {X 0,Y 607.889,Z 598.51,A -85,B 0,C 180,E1 27356.606,E2 27356.606} C_VEL
LIN {X 0,Y 607.905,Z 598.506,A -85,B 0,C 180,E1 27353.484,E2 27353.484} C_VEL
LIN {X 0,Y 607.889,Z 598.511,A -85,B 0,C 180,E1 27350.342,E2 27350.342} C_VEL
LIN {X 0,Y 607.908,Z 598.505,A -85,B 0,C 180,E1 27347.248,E2 27347.248} C_VEL
LIN {X 0,Y 607.886,Z 598.511,A -85,B 0,C 180,E1 27344.057,E2 27344.057} C_VEL
LIN {X 0,Y 607.906,Z 598.506,A -85,B 0,C 180,E1 27340.895,E2 27340.895} C_VEL
LIN {X 0,Y 607.885,Z 598.51,A -85,B 0,C 180,E1 27337.771,E2 27337.771} C_VEL
LIN {X 0,Y 607.909,Z 598.506,A -85,B 0,C 180,E1 27334.683,E2 27334.683} C_VEL
LIN {X 0,Y 607.884,Z 598.511,A -85,B 0,C 180,E1 27331.511,E2 27331.511} C_VEL
LIN {X 0,Y 607.907,Z 598.507,A -85,B 0,C 180,E1 27328.354,E2 27328.354} C_VEL
LIN {X 0,Y 607.881,Z 598.51,A -85,B 0,C 180,E1 27325.197,E2 27325.197} C_VEL
LIN {X 0,Y 607.907,Z 598.508,A -85,B 0,C 180,E1 27322.038,E2 27322.038} C_VEL
LIN {X 0,Y 607.881,Z 598.511,A -85,B 0,C 180,E1 27318.983,E2 27318.983} C_VEL
LIN {X 0,Y 607.913,Z 598.505,A -85,B 0,C 180,E1 27315.915,E2 27315.915} C_VEL
LIN {X 0,Y 607.882,Z 598.511,A -85,B 0,C 180,E1 27312.79,E2 27312.79} C_VEL
LIN {X 0,Y 607.912,Z 598.506,A -85,B 0,C 180,E1 27309.655,E2 27309.655} C_VEL
LIN {X 0,Y 607.878,Z 598.511,A -85,B 0,C 180,E1 27306.455,E2 27306.455} C_VEL
LIN {X 0,Y 607.912,Z 598.507,A -85,B 0,C 180,E1 27303.322,E2 27303.322} C_VEL
LIN {X 0,Y 607.912,Z 598.773,A -85,B 0,C 180,E1 27300.867,E2 27300.867} C_VEL
LIN {X 0,Y 607.918,Z 612.764,A -85,B 0,C 180,E1 27299.836,E2 27299.836} C_VEL
LIN {X 0,Y 607.913,Z 657.945,A -85,B 0,C 180,E1 27296.68,E2 27296.68} C_VEL
LIN {X 0,Y 607.851,Z 700.828,A -85,B 0,C 180,E1 27293.766,E2 27293.766} C_VEL
LIN {X 0,Y 607.895,Z 709.838,A -85,B 0,C 180,E1 27293.192,E2 27293.192} C_VEL
LIN {X 0,Y 607.914,Z 927.022,A -85,B 0,C 180,E1 27290.457,E2 27290.457} C_VEL
LIN {X 0,Y 607.916,Z 946.645,A -85,B 0,C 180,E1 27290.027,E2 27290.027} C_VEL
LIN {X 0,Y 607.915,Z 965.466,A -85,B 0,C 180,E1 27289.429,E2 27289.429} C_VEL
LIN {X 0,Y 607.916,Z 984.172,A -85,B 0,C 180,E1 27288.64,E2 27288.64} C_VEL
LIN {X 0,Y 607.918,Z 1001.543,A -85,B 0,C 180,E1 27287.714,E2 27287.714} C_VEL
LIN {X 0,Y 607.917,Z 1018.144,A -85,B 0,C 180,E1 27286.629,E2 27286.629} C_VEL
LIN {X 0,Y 607.915,Z 1033.664,A -85,B 0,C 180,E1 27285.404,E2 27285.404} C_VEL
LIN {X 0,Y 607.916,Z 1047.612,A -85,B 0,C 180,E1 27284.088,E2 27284.088} C_VEL
LIN {X 0,Y 607.914,Z 1060.52,A -85,B 0,C 180,E1 27282.635,E2 27282.635} C_VEL
LIN {X 0,Y 607.91,Z 1071.93,A -85,B 0,C 180,E1 27281.095,E2 27281.095} C_VEL
LIN {X 0,Y 607.913,Z 1081.846,A -85,B 0,C 180,E1 27279.466,E2 27279.466} C_VEL
LIN {X 0,Y 607.911,Z 1090.243,A -85,B 0,C 180,E1 27277.751,E2 27277.751} C_VEL
LIN {X 0,Y 607.909,Z 1096.733,A -85,B 0,C 180,E1 27276.042,E2 27276.042} C_VEL
LIN {X 0,Y 607.913,Z 1101.504,A -85,B 0,C 180,E1 27274.339,E2 27274.339} C_VEL
LIN {X 0,Y 607.908,Z 1104.775,A -85,B 0,C 180,E1 27272.545,E2 27272.545} C_VEL
LIN {X 0,Y 607.913,Z 1106.329,A -85,B 0,C 180,E1 27270.754,E2 27270.754} C_VEL
LIN {X 0,Y 607.906,Z 1106.195,A -85,B 0,C 180,E1 27268.963,E2 27268.963} C_VEL
LIN {X 0,Y 607.904,Z 1104.38,A -85,B 0,C 180,E1 27267.171,E2 27267.171} C_VEL
LIN {X 0,Y 607.912,Z 1100.776,A -85,B 0,C 180,E1 27265.353,E2 27265.353} C_VEL
LIN {X 0,Y 607.914,Z 1095.475,A -85,B 0,C 180,E1 27263.578,E2 27263.578} C_VEL
LIN {X 0,Y 607.914,Z 1088.596,A -85,B 0,C 180,E1 27261.868,E2 27261.868} C_VEL
LIN {X 0,Y 607.912,Z 1079.615,A -85,B 0,C 180,E1 27260.13,E2 27260.13} C_VEL
LIN {X 0,Y 607.914,Z 1069.317,A -85,B 0,C 180,E1 27258.52,E2 27258.52} C_VEL
LIN {X 0,Y 607.914,Z 1057.326,A -85,B 0,C 180,E1 27256.977,E2 27256.977} C_VEL
LIN {X 0,Y 607.913,Z 1044.232,A -85,B 0,C 180,E1 27255.571,E2 27255.571} C_VEL
LIN {X 0,Y 607.916,Z 1029.574,A -85,B 0,C 180,E1 27254.253,E2 27254.253} C_VEL
LIN {X 0,Y 607.918,Z 1013.879,A -85,B 0,C 180,E1 27253.075,E2 27253.075} C_VEL
LIN {X 0,Y 607.919,Z 997.167,A -85,B 0,C 180,E1 27252.038,E2 27252.038} C_VEL
LIN {X 0,Y 607.917,Z 979.411,A -85,B 0,C 180,E1 27251.144,E2 27251.144} C_VEL
LIN {X 0,Y 607.911,Z 961.4,A -85,B 0,C 180,E1 27250.43,E2 27250.43} C_VEL
LIN {X 0,Y 607.913,Z 943.468,A -85,B 0,C 180,E1 27249.894,E2 27249.894} C_VEL
LIN {X 0,Y 607.913,Z 925.335,A -85,B 0,C 180,E1 27249.517,E2 27249.517} C_VEL
LIN {X 0,Y 607.894,Z 709.32,A -85,B 0,C 180,E1 27246.796,E2 27246.796} C_VEL
LIN {X 0,Y 607.868,Z 667.126,A -85,B 0,C 180,E1 27243.948,E2 27243.948} C_VEL
LIN {X 0,Y 607.916,Z 624.243,A -85,B 0,C 180,E1 27240.974,E2 27240.974} C_VEL
LIN {X 0,Y 607.913,Z 598.881,A -85,B 0,C 180,E1 27239.154,E2 27239.154} C_VEL
LIN {X 0,Y 607.912,Z 598.504,A -85,B 0,C 180,E1 27238.685,E2 27238.685} C_VEL
LIN {X 0,Y 607.887,Z 598.513,A -85,B 0,C 180,E1 27235.541,E2 27235.541} C_VEL
LIN {X 0,Y 607.914,Z 598.504,A -85,B 0,C 180,E1 27232.277,E2 27232.277} C_VEL
LIN {X 0,Y 607.917,Z 598.514,A -85,B 0,C 180,E1 27228.985,E2 27228.985} C_VEL
LIN {X 0,Y 607.899,Z 598.506,A -85,B 0,C 180,E1 27225.782,E2 27225.782} C_VEL
LIN {X 0,Y 607.905,Z 598.512,A -85,B 0,C 180,E1 27222.66,E2 27222.66} C_VEL
LIN {X 0,Y 607.902,Z 598.506,A -85,B 0,C 180,E1 27219.52,E2 27219.52} C_VEL
LIN {X 0,Y 607.898,Z 598.512,A -85,B 0,C 180,E1 27216.425,E2 27216.425} C_VEL
LIN {X 0,Y 607.909,Z 598.505,A -85,B 0,C 180,E1 27213.322,E2 27213.322} C_VEL
LIN {X 0,Y 607.892,Z 598.512,A -85,B 0,C 180,E1 27210.219,E2 27210.219} C_VEL
LIN {X 0,Y 607.913,Z 598.505,A -85,B 0,C 180,E1 27207.103,E2 27207.103} C_VEL
LIN {X 0,Y 607.883,Z 598.512,A -85,B 0,C 180,E1 27203.971,E2 27203.971} C_VEL
LIN {X 0,Y 607.914,Z 598.506,A -85,B 0,C 180,E1 27200.809,E2 27200.809} C_VEL
LIN {X 0,Y 607.87,Z 598.511,A -85,B 0,C 180,E1 27197.617,E2 27197.617} C_VEL
LIN {X 0,Y 607.914,Z 598.509,A -85,B 0,C 180,E1 27194.477,E2 27194.477} C_VEL
LIN {X 0,Y 607.861,Z 598.512,A -85,B 0,C 180,E1 27191.375,E2 27191.375} C_VEL
LIN {X 0,Y 607.918,Z 598.508,A -85,B 0,C 180,E1 27188.322,E2 27188.322} C_VEL
LIN {X 0,Y 607.852,Z 598.515,A -85,B 0,C 180,E1 27185.19,E2 27185.19} C_VEL
LIN {X 0,Y 607.917,Z 598.782,A -85,B 0,C 180,E1 27183.937,E2 27183.937} C_VEL
LIN {X 0,Y 607.913,Z 626.496,A -85,B 0,C 180,E1 27180.848,E2 27180.848} C_VEL
LIN {X 0,Y 607.906,Z 656.892,A -85,B 0,C 180,E1 27177.549,E2 27177.549} C_VEL
LIN {X 0,Y 607.889,Z 664.253,A -85,B 0,C 180,E1 27176.761,E2 27176.761} C_VEL
LIN {X 0,Y 606.906,Z 669.513,A -85,B 0,C 180,E1 27176.23,E2 27176.23} C_VEL
LIN {X 0,Y 600.587,Z 684.739,A -85,B 0,C 180,E1 27174.794,E2 27174.794} C_VEL
LIN {X 0,Y 600.053,Z 688.507,A -85,B 0,C 180,E1 27174.406,E2 27174.406} C_VEL
LIN {X 0,Y 600.119,Z 693.103,A -85,B 0,C 180,E1 27173.966,E2 27173.966} C_VEL
LIN {X 0,Y 600.155,Z 832.667,A -85,B 0,C 180,E1 27172.241,E2 27172.241} C_VEL
LIN {X 0,Y 600.133,Z 849.614,A -85,B 0,C 180,E1 27171.84,E2 27171.84} C_VEL
LIN {X 0,Y 600.097,Z 864.201,A -85,B 0,C 180,E1 27171.327,E2 27171.327} C_VEL
LIN {X 0,Y 600.059,Z 879.364,A -85,B 0,C 180,E1 27170.602,E2 27170.602} C_VEL
LIN {X 0,Y 600.032,Z 893.508,A -85,B 0,C 180,E1 27169.729,E2 27169.729} C_VEL
LIN {X 0,Y 599.995,Z 906.556,A -85,B 0,C 180,E1 27168.708,E2 27168.708} C_VEL
LIN {X 0,Y 599.97,Z 918.22,A -85,B 0,C 180,E1 27167.576,E2 27167.576} C_VEL
LIN {X 0,Y 599.946,Z 928.645,A -85,B 0,C 180,E1 27166.311,E2 27166.311} C_VEL
LIN {X 0,Y 599.933,Z 937.68,A -85,B 0,C 180,E1 27164.93,E2 27164.93} C_VEL
LIN {X 0,Y 599.923,Z 944.694,A -85,B 0,C 180,E1 27163.541,E2 27163.541} C_VEL
LIN {X 0,Y 599.916,Z 950.27,A -85,B 0,C 180,E1 27162.041,E2 27162.041} C_VEL
LIN {X 0,Y 599.915,Z 954.068,A -85,B 0,C 180,E1 27160.529,E2 27160.529} C_VEL
LIN {X 0,Y 599.916,Z 956.1,A -85,B 0,C 180,E1 27158.961,E2 27158.961} C_VEL
LIN {X 0,Y 599.917,Z 956.367,A -85,B 0,C 180,E1 27157.356,E2 27157.356} C_VEL
LIN {X 0,Y 599.917,Z 954.761,A -85,B 0,C 180,E1 27155.795,E2 27155.795} C_VEL
LIN {X 0,Y 599.915,Z 951.309,A -85,B 0,C 180,E1 27154.214,E2 27154.214} C_VEL
LIN {X 0,Y 599.921,Z 946.175,A -85,B 0,C 180,E1 27152.72,E2 27152.72} C_VEL
LIN {X 0,Y 599.926,Z 938.941,A -85,B 0,C 180,E1 27151.206,E2 27151.206} C_VEL
LIN {X 0,Y 599.943,Z 930.679,A -85,B 0,C 180,E1 27149.879,E2 27149.879} C_VEL
LIN {X 0,Y 599.963,Z 920.226,A -85,B 0,C 180,E1 27148.558,E2 27148.558} C_VEL
LIN {X 0,Y 599.99,Z 909.181,A -85,B 0,C 180,E1 27147.434,E2 27147.434} C_VEL
LIN {X 0,Y 600.021,Z 896.677,A -85,B 0,C 180,E1 27146.41,E2 27146.41} C_VEL
LIN {X 0,Y 600.046,Z 882.644,A -85,B 0,C 180,E1 27145.49,E2 27145.49} C_VEL
LIN {X 0,Y 600.083,Z 867.612,A -85,B 0,C 180,E1 27144.73,E2 27144.73} C_VEL
LIN {X 0,Y 600.127,Z 851.545,A -85,B 0,C 180,E1 27144.127,E2 27144.127} C_VEL
LIN {X 0,Y 600.152,Z 835.497,A -85,B 0,C 180,E1 27143.722,E2 27143.722} C_VEL
LIN {X 0,Y 600.148,Z 811.855,A -85,B 0,C 180,E1 27143.391,E2 27143.391} C_VEL
LIN {X 0,Y 600.064,Z 692.613,A -85,B 0,C 180,E1 27141.924,E2 27141.924} C_VEL
LIN {X 0,Y 600.107,Z 663.372,A -85,B 0,C 180,E1 27138.8,E2 27138.8} C_VEL
LIN {X 0,Y 600.17,Z 634.117,A -85,B 0,C 180,E1 27135.596,E2 27135.596} C_VEL
LIN {X 0,Y 600.269,Z 605.78,A -85,B 0,C 180,E1 27132.424,E2 27132.424} C_VEL
LIN {X 0,Y 600.022,Z 599.925,A -85,B 0,C 180,E1 27131.738,E2 27131.738} C_VEL
LIN {X 0,Y 599.936,Z 599.507,A -85,B 0,C 180,E1 27131.553,E2 27131.553} C_VEL
LIN {X 0,Y 599.903,Z 599.503,A -85,B 0,C 180,E1 27128.684,E2 27128.684} C_VEL
LIN {X 0,Y 599.971,Z 599.5,A -85,B 0,C 180,E1 27125.564,E2 27125.564} C_VEL
LIN {X 0,Y 599.906,Z 599.501,A -85,B 0,C 180,E1 27122.504,E2 27122.504} C_VEL
LIN {X 0,Y 599.979,Z 599.501,A -85,B 0,C 180,E1 27119.447,E2 27119.447} C_VEL
LIN {X 0,Y 599.91,Z 599.501,A -85,B 0,C 180,E1 27116.317,E2 27116.317} C_VEL
LIN {X 0,Y 599.978,Z 599.502,A -85,B 0,C 180,E1 27113.264,E2 27113.264} C_VEL
LIN {X 0,Y 599.916,Z 599.499,A -85,B 0,C 180,E1 27110.182,E2 27110.182} C_VEL
LIN {X 0,Y 599.974,Z 599.503,A -85,B 0,C 180,E1 27107.156,E2 27107.156} C_VEL
LIN {X 0,Y 599.921,Z 599.5,A -85,B 0,C 180,E1 27103.985,E2 27103.985} C_VEL
LIN {X 0,Y 599.97,Z 599.503,A -85,B 0,C 180,E1 27100.952,E2 27100.952} C_VEL
LIN {X 0,Y 599.974,Z 599.741,A -85,B 0,C 180,E1 27099.206,E2 27099.206} C_VEL
LIN {X 0,Y 600.275,Z 603.734,A -85,B 0,C 180,E1 27098.719,E2 27098.719} C_VEL
LIN {X 0,Y 600.163,Z 632.03,A -85,B 0,C 180,E1 27095.545,E2 27095.545} C_VEL
LIN {X 0,Y 600.113,Z 660.812,A -85,B 0,C 180,E1 27092.387,E2 27092.387} C_VEL
LIN {X 0,Y 600.032,Z 690.1,A -85,B 0,C 180,E1 27089.236,E2 27089.236} C_VEL
LIN {X 0,Y 600.103,Z 693.188,A -85,B 0,C 180,E1 27088.965,E2 27088.965} C_VEL
LIN {X 0,Y 600.152,Z 832.733,A -85,B 0,C 180,E1 27087.24,E2 27087.24} C_VEL
LIN {X 0,Y 600.132,Z 849.641,A -85,B 0,C 180,E1 27086.84,E2 27086.84} C_VEL
LIN {X 0,Y 600.099,Z 864.318,A -85,B 0,C 180,E1 27086.322,E2 27086.322} C_VEL
LIN {X 0,Y 600.06,Z 879.309,A -85,B 0,C 180,E1 27085.604,E2 27085.604} C_VEL
LIN {X 0,Y 600.032,Z 893.318,A -85,B 0,C 180,E1 27084.742,E2 27084.742} C_VEL
LIN {X 0,Y 599.996,Z 906.256,A -85,B 0,C 180,E1 27083.734,E2 27083.734} C_VEL
LIN {X 0,Y 599.969,Z 918.361,A -85,B 0,C 180,E1 27082.561,E2 27082.561} C_VEL
LIN {X 0,Y 599.945,Z 928.884,A -85,B 0,C 180,E1 27081.277,E2 27081.277} C_VEL
LIN {X 0,Y 599.931,Z 937.725,A -85,B 0,C 180,E1 27079.922,E2 27079.922} C_VEL
LIN {X 0,Y 599.922,Z 944.776,A -85,B 0,C 180,E1 27078.52,E2 27078.52} C_VEL
LIN {X 0,Y 599.916,Z 950.405,A -85,B 0,C 180,E1 27076.997,E2 27076.997} C_VEL
LIN {X 0,Y 599.919,Z 954.08,A -85,B 0,C 180,E1 27075.523,E2 27075.523} C_VEL
LIN {X 0,Y 599.914,Z 956.116,A -85,B 0,C 180,E1 27073.939,E2 27073.939} C_VEL
LIN {X 0,Y 599.915,Z 956.362,A -85,B 0,C 180,E1 27072.342,E2 27072.342} C_VEL
LIN {X 0,Y 599.915,Z 954.657,A -85,B 0,C 180,E1 27070.731,E2 27070.731} C_VEL
LIN {X 0,Y 599.919,Z 951.288,A -85,B 0,C 180,E1 27069.207,E2 27069.207} C_VEL
LIN {X 0,Y 599.924,Z 946.38,A -85,B 0,C 180,E1 27067.77,E2 27067.77} C_VEL
LIN {X 0,Y 599.929,Z 939.54,A -85,B 0,C 180,E1 27066.318,E2 27066.318} C_VEL
LIN {X 0,Y 599.943,Z 931.22,A -85,B 0,C 180,E1 27064.956,E2 27064.956} C_VEL
LIN {X 0,Y 599.961,Z 921.335,A -85,B 0,C 180,E1 27063.686,E2 27063.686} C_VEL
LIN {X 0,Y 599.987,Z 909.991,A -85,B 0,C 180,E1 27062.509,E2 27062.509} C_VEL
LIN {X 0,Y 600.02,Z 897.943,A -85,B 0,C 180,E1 27061.504,E2 27061.504} C_VEL
LIN {X 0,Y 600.053,Z 883.771,A -85,B 0,C 180,E1 27060.557,E2 27060.557} C_VEL
LIN {X 0,Y 600.079,Z 869.718,A -85,B 0,C 180,E1 27059.823,E2 27059.823} C_VEL
LIN {X 0,Y 600.12,Z 854.856,A -85,B 0,C 180,E1 27059.237,E2 27059.237} C_VEL
LIN {X 0,Y 600.145,Z 838.386,A -85,B 0,C 180,E1 27058.78,E2 27058.78} C_VEL
LIN {X 0,Y 600.163,Z 820.785,A -85,B 0,C 180,E1 27058.5,E2 27058.5} C_VEL
LIN {X 0,Y 600.06,Z 692.616,A -85,B 0,C 180,E1 27056.924,E2 27056.924} C_VEL
LIN {X 0,Y 600.117,Z 662.804,A -85,B 0,C 180,E1 27053.739,E2 27053.739} C_VEL
LIN {X 0,Y 600.167,Z 634.15,A -85,B 0,C 180,E1 27050.6,E2 27050.6} C_VEL
LIN {X 0,Y 600.273,Z 604.849,A -85,B 0,C 180,E1 27047.318,E2 27047.318} C_VEL
LIN {X 0,Y 600.025,Z 599.92,A -85,B 0,C 180,E1 27046.736,E2 27046.736} C_VEL
LIN {X 0,Y 599.961,Z 599.503,A -85,B 0,C 180,E1 27046.374,E2 27046.374} C_VEL
LIN {X 0,Y 599.956,Z 599.501,A -85,B 0,C 180,E1 27043.232,E2 27043.232} C_VEL
LIN {X 0,Y 599.963,Z 599.495,A -85,B 0,C 180,E1 27040.037,E2 27040.037} C_VEL
LIN {X 0,Y 599.97,Z 599.503,A -85,B 0,C 180,E1 27036.747,E2 27036.747} C_VEL
LIN {X 0,Y 599.97,Z 599.493,A -85,B 0,C 180,E1 27033.364,E2 27033.364} C_VEL
LIN {X 0,Y 599.962,Z 599.501,A -85,B 0,C 180,E1 27030.108,E2 27030.108} C_VEL
LIN {X 0,Y 599.962,Z 599.495,A -85,B 0,C 180,E1 27026.926,E2 27026.926} C_VEL
LIN {X 0,Y 599.958,Z 599.5,A -85,B 0,C 180,E1 27023.785,E2 27023.785} C_VEL
LIN {X 0,Y 599.961,Z 599.496,A -85,B 0,C 180,E1 27020.588,E2 27020.588} C_VEL
LIN {X 0,Y 599.955,Z 599.5,A -85,B 0,C 180,E1 27017.457,E2 27017.457} C_VEL
LIN {X 0,Y 599.961,Z 599.496,A -85,B 0,C 180,E1 27014.279,E2 27014.279} C_VEL
LIN {X 0,Y 599.953,Z 599.498,A -85,B 0,C 180,E1 27011.147,E2 27011.147} C_VEL
LIN {X 0,Y 599.961,Z 599.497,A -85,B 0,C 180,E1 27007.951,E2 27007.951} C_VEL
LIN {X 0,Y 599.951,Z 599.499,A -85,B 0,C 180,E1 27004.876,E2 27004.876} C_VEL
LIN {X 0,Y 599.963,Z 599.497,A -85,B 0,C 180,E1 27001.719,E2 27001.719} C_VEL
LIN {X 0,Y 599.949,Z 599.499,A -85,B 0,C 180,E1 26998.568,E2 26998.568} C_VEL
LIN {X 0,Y 599.963,Z 599.496,A -85,B 0,C 180,E1 26995.412,E2 26995.412} C_VEL
LIN {X 0,Y 599.948,Z 599.498,A -85,B 0,C 180,E1 26992.338,E2 26992.338} C_VEL
LIN {X 0,Y 599.966,Z 599.495,A -85,B 0,C 180,E1 26989.243,E2 26989.243} C_VEL
LIN {X 0,Y 599.948,Z 599.499,A -85,B 0,C 180,E1 26986.114,E2 26986.114} C_VEL
LIN {X 0,Y 599.969,Z 599.495,A -85,B 0,C 180,E1 26983.044,E2 26983.044} C_VEL
LIN {X 0,Y 599.946,Z 599.499,A -85,B 0,C 180,E1 26979.819,E2 26979.819} C_VEL
LIN {X 0,Y 599.967,Z 599.496,A -85,B 0,C 180,E1 26976.672,E2 26976.672} C_VEL
LIN {X 0,Y 599.944,Z 599.498,A -85,B 0,C 180,E1 26973.503,E2 26973.503} C_VEL
LIN {X 0,Y 599.967,Z 599.498,A -85,B 0,C 180,E1 26970.333,E2 26970.333} C_VEL
LIN {X 0,Y 599.942,Z 599.499,A -85,B 0,C 180,E1 26967.205,E2 26967.205} C_VEL
LIN {X 0,Y 599.968,Z 599.497,A -85,B 0,C 180,E1 26964.083,E2 26964.083} C_VEL
LIN {X 0,Y 599.941,Z 599.499,A -85,B 0,C 180,E1 26960.952,E2 26960.952} C_VEL
LIN {X 0,Y 599.969,Z 599.498,A -85,B 0,C 180,E1 26957.809,E2 26957.809} C_VEL
LIN {X 0,Y 599.939,Z 599.499,A -85,B 0,C 180,E1 26954.693,E2 26954.693} C_VEL
LIN {X 0,Y 599.97,Z 599.498,A -85,B 0,C 180,E1 26951.55,E2 26951.55} C_VEL
LIN {X 0,Y 599.938,Z 599.499,A -85,B 0,C 180,E1 26948.436,E2 26948.436} C_VEL
LIN {X 0,Y 599.971,Z 599.498,A -85,B 0,C 180,E1 26945.329,E2 26945.329} C_VEL
LIN {X 0,Y 599.935,Z 599.493,A -85,B 0,C 180,E1 26942.152,E2 26942.152} C_VEL
LIN {X 0,Y 600.016,Z 599.789,A -85,B 0,C 180,E1 26941.24,E2 26941.24} C_VEL
LIN {X 0,Y 600.693,Z 602.809,A -85,B 0,C 180,E1 26940.953,E2 26940.953} C_VEL
LIN {X 0,Y 600.517,Z 644.926,A -85,B 0,C 180,E1 26937.949,E2 26937.949} C_VEL
LIN {X 0,Y 600.4,Z 690.107,A -85,B 0,C 180,E1 26934.813,E2 26934.813} C_VEL
LIN {X 0,Y 600.428,Z 709.849,A -85,B 0,C 180,E1 26933.498,E2 26933.498} C_VEL
LIN {X 0,Y 600.407,Z 927.531,A -85,B 0,C 180,E1 26930.715,E2 26930.715} C_VEL
LIN {X 0,Y 600.371,Z 946.852,A -85,B 0,C 180,E1 26930.283,E2 26930.283} C_VEL
LIN {X 0,Y 600.326,Z 964.794,A -85,B 0,C 180,E1 26929.71,E2 26929.71} C_VEL
LIN {X 0,Y 600.275,Z 982.783,A -85,B 0,C 180,E1 26928.954,E2 26928.954} C_VEL
LIN {X 0,Y 600.21,Z 1000.725,A -85,B 0,C 180,E1 26928,E2 26928} C_VEL
LIN {X 0,Y 600.144,Z 1017.477,A -85,B 0,C 180,E1 26926.901,E2 26926.901} C_VEL
LIN {X 0,Y 600.079,Z 1033.112,A -85,B 0,C 180,E1 26925.66,E2 26925.66} C_VEL
LIN {X 0,Y 600.03,Z 1046.686,A -85,B 0,C 180,E1 26924.376,E2 26924.376} C_VEL
LIN {X 0,Y 599.987,Z 1059.747,A -85,B 0,C 180,E1 26922.903,E2 26922.903} C_VEL
LIN {X 0,Y 599.96,Z 1071.292,A -85,B 0,C 180,E1 26921.341,E2 26921.341} C_VEL
LIN {X 0,Y 599.932,Z 1081.329,A -85,B 0,C 180,E1 26919.69,E2 26919.69} C_VEL
LIN {X 0,Y 599.926,Z 1089.432,A -85,B 0,C 180,E1 26918.047,E2 26918.047} C_VEL
LIN {X 0,Y 599.921,Z 1096.129,A -85,B 0,C 180,E1 26916.315,E2 26916.315} C_VEL
LIN {X 0,Y 599.913,Z 1101.299,A -85,B 0,C 180,E1 26914.493,E2 26914.493} C_VEL
LIN {X 0,Y 599.904,Z 1104.663,A -85,B 0,C 180,E1 26912.675,E2 26912.675} C_VEL
LIN {X 0,Y 599.911,Z 1106.306,A -85,B 0,C 180,E1 26910.859,E2 26910.859} C_VEL
LIN {X 0,Y 599.909,Z 1106.262,A -85,B 0,C 180,E1 26909.045,E2 26909.045} C_VEL
LIN {X 0,Y 599.903,Z 1104.536,A -85,B 0,C 180,E1 26907.229,E2 26907.229} C_VEL
LIN {X 0,Y 599.913,Z 1101.086,A -85,B 0,C 180,E1 26905.411,E2 26905.411} C_VEL
LIN {X 0,Y 599.919,Z 1095.819,A -85,B 0,C 180,E1 26903.588,E2 26903.588} C_VEL
LIN {X 0,Y 599.929,Z 1088.596,A -85,B 0,C 180,E1 26901.759,E2 26901.759} C_VEL
LIN {X 0,Y 599.945,Z 1079.737,A -85,B 0,C 180,E1 26900.019,E2 26900.019} C_VEL
LIN {X 0,Y 599.965,Z 1069.316,A -85,B 0,C 180,E1 26898.366,E2 26898.366} C_VEL
LIN {X 0,Y 600.004,Z 1057.326,A -85,B 0,C 180,E1 26896.803,E2 26896.803} C_VEL
LIN {X 0,Y 600.044,Z 1044.232,A -85,B 0,C 180,E1 26895.377,E2 26895.377} C_VEL
LIN {X 0,Y 600.096,Z 1029.576,A -85,B 0,C 180,E1 26894.043,E2 26894.043} C_VEL
LIN {X 0,Y 600.156,Z 1013.881,A -85,B 0,C 180,E1 26892.849,E2 26892.849} C_VEL
LIN {X 0,Y 600.219,Z 997.17,A -85,B 0,C 180,E1 26891.799,E2 26891.799} C_VEL
LIN {X 0,Y 600.279,Z 979.414,A -85,B 0,C 180,E1 26890.895,E2 26890.895} C_VEL
LIN {X 0,Y 600.33,Z 961.11,A -85,B 0,C 180,E1 26890.163,E2 26890.163} C_VEL
LIN {X 0,Y 600.38,Z 942.095,A -85,B 0,C 180,E1 26889.597,E2 26889.597} C_VEL
LIN {X 0,Y 600.417,Z 922.871,A -85,B 0,C 180,E1 26889.213,E2 26889.213} C_VEL
LIN {X 0,Y 600.423,Z 709.72,A -85,B 0,C 180,E1 26886.497,E2 26886.497} C_VEL
LIN {X 0,Y 600.431,Z 669.423,A -85,B 0,C 180,E1 26883.76,E2 26883.76} C_VEL
LIN {X 0,Y 600.612,Z 626.234,A -85,B 0,C 180,E1 26880.729,E2 26880.729} C_VEL
LIN {X 0,Y 600.569,Z 601.691,A -85,B 0,C 180,E1 26878.959,E2 26878.959} C_VEL
LIN {X 0,Y 599.988,Z 599.609,A -85,B 0,C 180,E1 26878.718,E2 26878.718} C_VEL
LIN {X 0,Y 599.947,Z 599.503,A -85,B 0,C 180,E1 26875.584,E2 26875.584} C_VEL
LIN {X 0,Y 599.977,Z 599.494,A -85,B 0,C 180,E1 26872.294,E2 26872.294} C_VEL
LIN {X 0,Y 599.977,Z 599.503,A -85,B 0,C 180,E1 26868.959,E2 26868.959} C_VEL
LIN {X 0,Y 599.957,Z 599.495,A -85,B 0,C 180,E1 26865.71,E2 26865.71} C_VEL
LIN {X 0,Y 599.961,Z 599.5,A -85,B 0,C 180,E1 26862.556,E2 26862.556} C_VEL
LIN {X 0,Y 599.959,Z 599.497,A -85,B 0,C 180,E1 26859.35,E2 26859.35} C_VEL
LIN {X 0,Y 599.953,Z 599.499,A -85,B 0,C 180,E1 26856.233,E2 26856.233} C_VEL
LIN {X 0,Y 599.964,Z 599.497,A -85,B 0,C 180,E1 26853.135,E2 26853.135} C_VEL
LIN {X 0,Y 599.945,Z 599.499,A -85,B 0,C 180,E1 26849.998,E2 26849.998} C_VEL
LIN {X 0,Y 599.968,Z 599.498,A -85,B 0,C 180,E1 26846.848,E2 26846.848} C_VEL
LIN {X 0,Y 599.938,Z 599.499,A -85,B 0,C 180,E1 26843.786,E2 26843.786} C_VEL
LIN {X 0,Y 599.972,Z 599.497,A -85,B 0,C 180,E1 26840.689,E2 26840.689} C_VEL
LIN {X 0,Y 599.93,Z 599.5,A -85,B 0,C 180,E1 26837.557,E2 26837.557} C_VEL
LIN {X 0,Y 599.976,Z 599.498,A -85,B 0,C 180,E1 26834.476,E2 26834.476} C_VEL
LIN {X 0,Y 599.922,Z 599.501,A -85,B 0,C 180,E1 26831.342,E2 26831.342} C_VEL
LIN {X 0,Y 599.978,Z 599.499,A -85,B 0,C 180,E1 26828.24,E2 26828.24} C_VEL
LIN {X 0,Y 599.914,Z 599.507,A -85,B 0,C 180,E1 26825.163,E2 26825.163} C_VEL
LIN {X 0,Y 600.013,Z 599.769,A -85,B 0,C 180,E1 26824.193,E2 26824.193} C_VEL
LIN {X 0,Y 600.272,Z 605.366,A -85,B 0,C 180,E1 26823.533,E2 26823.533} C_VEL
LIN {X 0,Y 600.182,Z 635.222,A -85,B 0,C 180,E1 26820.191,E2 26820.191} C_VEL
LIN {X 0,Y 600.1,Z 664.026,A -85,B 0,C 180,E1 26817.039,E2 26817.039} C_VEL
LIN {X 0,Y 600.053,Z 688.507,A -85,B 0,C 180,E1 26814.406,E2 26814.406} C_VEL
LIN {X 0,Y 599.512,Z 691.848,A -85,B 0,C 180,E1 26814.169,E2 26814.169} C_VEL
LIN {X 0,Y 597.912,Z 696.763,A -85,B 0,C 180,E1 26814.021,E2 26814.021} C_VEL
LIN {X 0,Y 594.315,Z 707.569,A -85,B 0,C 180,E1 26813.945,E2 26813.945} C_VEL
LIN {X 0,Y 592.654,Z 718.018,A -85,B 0,C 180,E1 26813.862,E2 26813.862} C_VEL
LIN {X 0,Y 592.499,Z 722.706,A -85,B 0,C 180,E1 26813.808,E2 26813.808} C_VEL
LIN {X 0,Y 592.397,Z 832.706,A -85,B 0,C 180,E1 26812.432,E2 26812.432} C_VEL
LIN {X 0,Y 592.352,Z 849.757,A -85,B 0,C 180,E1 26812.022,E2 26812.022} C_VEL
LIN {X 0,Y 592.277,Z 865.365,A -85,B 0,C 180,E1 26811.456,E2 26811.456} C_VEL
LIN {X 0,Y 592.208,Z 880.29,A -85,B 0,C 180,E1 26810.721,E2 26810.721} C_VEL
LIN {X 0,Y 592.144,Z 894.224,A -85,B 0,C 180,E1 26809.837,E2 26809.837} C_VEL
LIN {X 0,Y 592.075,Z 907.144,A -85,B 0,C 180,E1 26808.802,E2 26808.802} C_VEL
LIN {X 0,Y 592.018,Z 919.049,A -85,B 0,C 180,E1 26807.614,E2 26807.614} C_VEL
LIN {X 0,Y 591.974,Z 929.384,A -85,B 0,C 180,E1 26806.322,E2 26806.322} C_VEL
LIN {X 0,Y 591.945,Z 938.257,A -85,B 0,C 180,E1 26804.922,E2 26804.922} C_VEL
LIN {X 0,Y 591.928,Z 945.544,A -85,B 0,C 180,E1 26803.413,E2 26803.413} C_VEL
LIN {X 0,Y 591.916,Z 950.9,A -85,B 0,C 180,E1 26801.892,E2 26801.892} C_VEL
LIN {X 0,Y 591.914,Z 954.417,A -85,B 0,C 180,E1 26800.357,E2 26800.357} C_VEL
LIN {X 0,Y 591.912,Z 956.285,A -85,B 0,C 180,E1 26798.704,E2 26798.704} C_VEL
LIN {X 0,Y 591.915,Z 956.239,A -85,B 0,C 180,E1 26797.138,E2 26797.138} C_VEL
LIN {X 0,Y 591.914,Z 954.417,A -85,B 0,C 180,E1 26795.553,E2 26795.553} C_VEL
LIN {X 0,Y 591.917,Z 950.789,A -85,B 0,C 180,E1 26793.982,E2 26793.982} C_VEL
LIN {X 0,Y 591.925,Z 945.264,A -85,B 0,C 180,E1 26792.43,E2 26792.43} C_VEL
LIN {X 0,Y 591.944,Z 938.339,A -85,B 0,C 180,E1 26791.002,E2 26791.002} C_VEL
LIN {X 0,Y 591.973,Z 929.947,A -85,B 0,C 180,E1 26789.666,E2 26789.666} C_VEL
LIN {X 0,Y 592.018,Z 919.221,A -85,B 0,C 180,E1 26788.315,E2 26788.315} C_VEL
LIN {X 0,Y 592.073,Z 907.458,A -85,B 0,C 180,E1 26787.136,E2 26787.136} C_VEL
LIN {X 0,Y 592.141,Z 894.311,A -85,B 0,C 180,E1 26786.08,E2 26786.08} C_VEL
LIN {X 0,Y 592.208,Z 880.544,A -85,B 0,C 180,E1 26785.203,E2 26785.203} C_VEL
LIN {X 0,Y 592.275,Z 865.499,A -85,B 0,C 180,E1 26784.459,E2 26784.459} C_VEL
LIN {X 0,Y 592.351,Z 849.891,A -85,B 0,C 180,E1 26783.891,E2 26783.891} C_VEL
LIN {X 0,Y 592.394,Z 832.987,A -85,B 0,C 180,E1 26783.484,E2 26783.484} C_VEL
LIN {X 0,Y 592.438,Z 761.161,A -85,B 0,C 180,E1 26782.574,E2 26782.574} C_VEL
LIN {X 0,Y 592.282,Z 693.262,A -85,B 0,C 180,E1 26781.73,E2 26781.73} C_VEL
LIN {X 0,Y 592.191,Z 690.769,A -85,B 0,C 180,E1 26781.524,E2 26781.524} C_VEL
LIN {X 0,Y 592.331,Z 662.108,A -85,B 0,C 180,E1 26778.4,E2 26778.4} C_VEL
LIN {X 0,Y 592.474,Z 631.227,A -85,B 0,C 180,E1 26774.965,E2 26774.965} C_VEL
LIN {X 0,Y 592.646,Z 603.259,A -85,B 0,C 180,E1 26771.78,E2 26771.78} C_VEL
LIN {X 0,Y 591.986,Z 600.538,A -85,B 0,C 180,E1 26771.381,E2 26771.381} C_VEL
LIN {X 0,Y 591.969,Z 600.493,A -85,B 0,C 180,E1 26768.553,E2 26768.553} C_VEL
LIN {X 0,Y 592,Z 600.49,A -85,B 0,C 180,E1 26765.284,E2 26765.284} C_VEL
LIN {X 0,Y 591.971,Z 600.49,A -85,B 0,C 180,E1 26762.373,E2 26762.373} C_VEL
LIN {X 0,Y 592.021,Z 600.487,A -85,B 0,C 180,E1 26759.172,E2 26759.172} C_VEL
LIN {X 0,Y 591.974,Z 600.49,A -85,B 0,C 180,E1 26756.158,E2 26756.158} C_VEL
LIN {X 0,Y 592.029,Z 600.487,A -85,B 0,C 180,E1 26752.963,E2 26752.963} C_VEL
LIN {X 0,Y 591.979,Z 600.488,A -85,B 0,C 180,E1 26749.949,E2 26749.949} C_VEL
LIN {X 0,Y 592.036,Z 600.484,A -85,B 0,C 180,E1 26746.748,E2 26746.748} C_VEL
LIN {X 0,Y 591.984,Z 600.491,A -85,B 0,C 180,E1 26743.678,E2 26743.678} C_VEL
LIN {X 0,Y 592.037,Z 600.485,A -85,B 0,C 180,E1 26740.51,E2 26740.51} C_VEL
LIN {X 0,Y 592.025,Z 600.764,A -85,B 0,C 180,E1 26739.478,E2 26739.478} C_VEL
LIN {X 0,Y 592.649,Z 604.165,A -85,B 0,C 180,E1 26739.027,E2 26739.027} C_VEL
LIN {X 0,Y 592.465,Z 631.553,A -85,B 0,C 180,E1 26735.909,E2 26735.909} C_VEL
LIN {X 0,Y 592.316,Z 659.43,A -85,B 0,C 180,E1 26732.806,E2 26732.806} C_VEL
LIN {X 0,Y 592.215,Z 687.769,A -85,B 0,C 180,E1 26729.71,E2 26729.71} C_VEL
LIN {X 0,Y 592.232,Z 692.968,A -85,B 0,C 180,E1 26729.19,E2 26729.19} C_VEL
LIN {X 0,Y 592.497,Z 702.789,A -85,B 0,C 180,E1 26729.054,E2 26729.054} C_VEL
LIN {X 0,Y 592.394,Z 832.756,A -85,B 0,C 180,E1 26727.431,E2 26727.431} C_VEL
LIN {X 0,Y 592.352,Z 849.666,A -85,B 0,C 180,E1 26727.025,E2 26727.025} C_VEL
LIN {X 0,Y 592.282,Z 865.104,A -85,B 0,C 180,E1 26726.468,E2 26726.468} C_VEL
LIN {X 0,Y 592.21,Z 879.939,A -85,B 0,C 180,E1 26725.74,E2 26725.74} C_VEL
LIN {X 0,Y 592.147,Z 893.829,A -85,B 0,C 180,E1 26724.866,E2 26724.866} C_VEL
LIN {X 0,Y 592.073,Z 907.201,A -85,B 0,C 180,E1 26723.796,E2 26723.796} C_VEL
LIN {X 0,Y 592.019,Z 918.953,A -85,B 0,C 180,E1 26722.626,E2 26722.626} C_VEL
LIN {X 0,Y 591.973,Z 929.139,A -85,B 0,C 180,E1 26721.355,E2 26721.355} C_VEL
LIN {X 0,Y 591.946,Z 937.932,A -85,B 0,C 180,E1 26719.981,E2 26719.981} C_VEL
LIN {X 0,Y 591.926,Z 945.162,A -85,B 0,C 180,E1 26718.503,E2 26718.503} C_VEL
LIN {X 0,Y 591.918,Z 950.514,A -85,B 0,C 180,E1 26717.017,E2 26717.017} C_VEL
LIN {X 0,Y 591.92,Z 954.144,A -85,B 0,C 180,E1 26715.523,E2 26715.523} C_VEL
LIN {X 0,Y 591.914,Z 956.14,A -85,B 0,C 180,E1 26713.917,E2 26713.917} C_VEL
LIN {X 0,Y 591.914,Z 956.346,A -85,B 0,C 180,E1 26712.299,E2 26712.299} C_VEL
LIN {X 0,Y 591.914,Z 954.601,A -85,B 0,C 180,E1 26710.666,E2 26710.666} C_VEL
LIN {X 0,Y 591.922,Z 951.102,A -85,B 0,C 180,E1 26709.086,E2 26709.086} C_VEL
LIN {X 0,Y 591.925,Z 945.79,A -85,B 0,C 180,E1 26707.558,E2 26707.558} C_VEL
LIN {X 0,Y 591.943,Z 938.532,A -85,B 0,C 180,E1 26706.038,E2 26706.038} C_VEL
LIN {X 0,Y 591.973,Z 929.749,A -85,B 0,C 180,E1 26704.64,E2 26704.64} C_VEL
LIN {X 0,Y 592.016,Z 919.131,A -85,B 0,C 180,E1 26703.305,E2 26703.305} C_VEL
LIN {X 0,Y 592.071,Z 907.76,A -85,B 0,C 180,E1 26702.164,E2 26702.164} C_VEL
LIN {X 0,Y 592.142,Z 894.435,A -85,B 0,C 180,E1 26701.088,E2 26701.088} C_VEL
LIN {X 0,Y 592.212,Z 880.578,A -85,B 0,C 180,E1 26700.206,E2 26700.206} C_VEL
LIN {X 0,Y 592.274,Z 865.514,A -85,B 0,C 180,E1 26699.46,E2 26699.46} C_VEL
LIN {X 0,Y 592.351,Z 849.971,A -85,B 0,C 180,E1 26698.894,E2 26698.894} C_VEL
LIN {X 0,Y 592.395,Z 833.216,A -85,B 0,C 180,E1 26698.488,E2 26698.488} C_VEL
LIN {X 0,Y 592.429,Z 780.023,A -85,B 0,C 180,E1 26697.806,E2 26697.806} C_VEL
LIN {X 0,Y 592.313,Z 693.475,A -85,B 0,C 180,E1 26696.734,E2 26696.734} C_VEL
LIN {X 0,Y 592.194,Z 691.512,A -85,B 0,C 180,E1 26696.605,E2 26696.605} C_VEL
LIN {X 0,Y 592.321,Z 662.343,A -85,B 0,C 180,E1 26693.425,E2 26693.425} C_VEL
LIN {X 0,Y 592.458,Z 633.651,A -85,B 0,C 180,E1 26690.237,E2 26690.237} C_VEL
LIN {X 0,Y 592.636,Z 605.437,A -85,B 0,C 180,E1 26687.031,E2 26687.031} C_VEL
LIN {X 0,Y 592.351,Z 602.002,A -85,B 0,C 180,E1 26686.607,E2 26686.607} C_VEL
LIN {X 0,Y 592.043,Z 600.638,A -85,B 0,C 180,E1 26686.382,E2 26686.382} C_VEL
LIN {X 0,Y 592.021,Z 600.492,A -85,B 0,C 180,E1 26683.157,E2 26683.157} C_VEL
LIN {X 0,Y 592.04,Z 600.481,A -85,B 0,C 180,E1 26679.797,E2 26679.797} C_VEL
LIN {X 0,Y 592.029,Z 600.492,A -85,B 0,C 180,E1 26676.476,E2 26676.476} C_VEL
LIN {X 0,Y 592.022,Z 600.484,A -85,B 0,C 180,E1 26673.175,E2 26673.175} C_VEL
LIN {X 0,Y 592.018,Z 600.488,A -85,B 0,C 180,E1 26669.957,E2 26669.957} C_VEL
LIN {X 0,Y 592.02,Z 600.486,A -85,B 0,C 180,E1 26666.804,E2 26666.804} C_VEL
LIN {X 0,Y 592.018,Z 600.488,A -85,B 0,C 180,E1 26663.701,E2 26663.701} C_VEL
LIN {X 0,Y 592.022,Z 600.485,A -85,B 0,C 180,E1 26660.566,E2 26660.566} C_VEL
LIN {X 0,Y 592.016,Z 600.488,A -85,B 0,C 180,E1 26657.394,E2 26657.394} C_VEL
LIN {X 0,Y 592.021,Z 600.485,A -85,B 0,C 180,E1 26654.206,E2 26654.206} C_VEL
LIN {X 0,Y 592.014,Z 600.485,A -85,B 0,C 180,E1 26651.002,E2 26651.002} C_VEL
LIN {X 0,Y 592.025,Z 600.488,A -85,B 0,C 180,E1 26647.765,E2 26647.765} C_VEL
LIN {X 0,Y 592.016,Z 600.484,A -85,B 0,C 180,E1 26644.553,E2 26644.553} C_VEL
LIN {X 0,Y 592.033,Z 600.492,A -85,B 0,C 180,E1 26641.258,E2 26641.258} C_VEL
LIN {X 0,Y 592.034,Z 600.482,A -85,B 0,C 180,E1 26637.871,E2 26637.871} C_VEL
LIN {X 0,Y 592.015,Z 600.489,A -85,B 0,C 180,E1 26634.573,E2 26634.573} C_VEL
LIN {X 0,Y 592.027,Z 600.484,A -85,B 0,C 180,E1 26631.355,E2 26631.355} C_VEL
LIN {X 0,Y 592.011,Z 600.488,A -85,B 0,C 180,E1 26628.208,E2 26628.208} C_VEL
LIN {X 0,Y 592.026,Z 600.484,A -85,B 0,C 180,E1 26625.024,E2 26625.024} C_VEL
LIN {X 0,Y 592.008,Z 600.486,A -85,B 0,C 180,E1 26621.895,E2 26621.895} C_VEL
LIN {X 0,Y 592.027,Z 600.486,A -85,B 0,C 180,E1 26618.709,E2 26618.709} C_VEL
LIN {X 0,Y 592.005,Z 600.487,A -85,B 0,C 180,E1 26615.552,E2 26615.552} C_VEL
LIN {X 0,Y 592.028,Z 600.487,A -85,B 0,C 180,E1 26612.326,E2 26612.326} C_VEL
LIN {X 0,Y 592.004,Z 600.486,A -85,B 0,C 180,E1 26609.22,E2 26609.22} C_VEL
LIN {X 0,Y 592.028,Z 600.489,A -85,B 0,C 180,E1 26606.02,E2 26606.02} C_VEL
LIN {X 0,Y 592.004,Z 600.486,A -85,B 0,C 180,E1 26602.861,E2 26602.861} C_VEL
LIN {X 0,Y 592.032,Z 600.49,A -85,B 0,C 180,E1 26599.697,E2 26599.697} C_VEL
LIN {X 0,Y 592.003,Z 600.485,A -85,B 0,C 180,E1 26596.572,E2 26596.572} C_VEL
LIN {X 0,Y 592.034,Z 600.49,A -85,B 0,C 180,E1 26593.422,E2 26593.422} C_VEL
LIN {X 0,Y 592.003,Z 600.486,A -85,B 0,C 180,E1 26590.235,E2 26590.235} C_VEL
LIN {X 0,Y 592.034,Z 600.493,A -85,B 0,C 180,E1 26586.958,E2 26586.958} C_VEL
LIN {X 0,Y 592.015,Z 600.488,A -85,B 0,C 180,E1 26583.755,E2 26583.755} C_VEL
LIN {X 0,Y 592.047,Z 600.71,A -85,B 0,C 180,E1 26581.648,E2 26581.648} C_VEL
LIN {X 0,Y 593.478,Z 605.106,A -85,B 0,C 180,E1 26581.202,E2 26581.202} C_VEL
LIN {X 0,Y 593.163,Z 647.224,A -85,B 0,C 180,E1 26578.163,E2 26578.163} C_VEL
LIN {X 0,Y 592.905,Z 692.404,A -85,B 0,C 180,E1 26574.988,E2 26574.988} C_VEL
LIN {X 0,Y 592.843,Z 709.485,A -85,B 0,C 180,E1 26573.824,E2 26573.824} C_VEL
LIN {X 0,Y 593.202,Z 715.116,A -85,B 0,C 180,E1 26573.729,E2 26573.729} C_VEL
LIN {X 0,Y 592.919,Z 927.531,A -85,B 0,C 180,E1 26570.989,E2 26570.989} C_VEL
LIN {X 0,Y 592.842,Z 946.851,A -85,B 0,C 180,E1 26570.552,E2 26570.552} C_VEL
LIN {X 0,Y 592.752,Z 964.795,A -85,B 0,C 180,E1 26569.973,E2 26569.973} C_VEL
LIN {X 0,Y 592.641,Z 982.784,A -85,B 0,C 180,E1 26569.207,E2 26569.207} C_VEL
LIN {X 0,Y 592.513,Z 1000.723,A -85,B 0,C 180,E1 26568.242,E2 26568.242} C_VEL
LIN {X 0,Y 592.383,Z 1017.475,A -85,B 0,C 180,E1 26567.129,E2 26567.129} C_VEL
LIN {X 0,Y 592.257,Z 1033.11,A -85,B 0,C 180,E1 26565.872,E2 26565.872} C_VEL
LIN {X 0,Y 592.159,Z 1046.686,A -85,B 0,C 180,E1 26564.571,E2 26564.571} C_VEL
LIN {X 0,Y 592.071,Z 1059.748,A -85,B 0,C 180,E1 26563.079,E2 26563.079} C_VEL
LIN {X 0,Y 592.01,Z 1071.293,A -85,B 0,C 180,E1 26561.495,E2 26561.495} C_VEL
LIN {X 0,Y 591.959,Z 1081.33,A -85,B 0,C 180,E1 26559.822,E2 26559.822} C_VEL
LIN {X 0,Y 591.939,Z 1089.432,A -85,B 0,C 180,E1 26558.157,E2 26558.157} C_VEL
LIN {X 0,Y 591.924,Z 1096.129,A -85,B 0,C 180,E1 26556.401,E2 26556.401} C_VEL
LIN {X 0,Y 591.914,Z 1101.299,A -85,B 0,C 180,E1 26554.553,E2 26554.553} C_VEL
LIN {X 0,Y 591.904,Z 1104.662,A -85,B 0,C 180,E1 26552.711,E2 26552.711} C_VEL
LIN {X 0,Y 591.912,Z 1106.306,A -85,B 0,C 180,E1 26550.871,E2 26550.871} C_VEL
LIN {X 0,Y 591.909,Z 1106.262,A -85,B 0,C 180,E1 26549.032,E2 26549.032} C_VEL
LIN {X 0,Y 591.905,Z 1104.536,A -85,B 0,C 180,E1 26547.192,E2 26547.192} C_VEL
LIN {X 0,Y 591.916,Z 1100.936,A -85,B 0,C 180,E1 26545.288,E2 26545.288} C_VEL
LIN {X 0,Y 591.923,Z 1095.819,A -85,B 0,C 180,E1 26543.501,E2 26543.501} C_VEL
LIN {X 0,Y 591.947,Z 1088.595,A -85,B 0,C 180,E1 26541.647,E2 26541.647} C_VEL
LIN {X 0,Y 591.979,Z 1079.737,A -85,B 0,C 180,E1 26539.883,E2 26539.883} C_VEL
LIN {X 0,Y 592.022,Z 1069.315,A -85,B 0,C 180,E1 26538.208,E2 26538.208} C_VEL
LIN {X 0,Y 592.094,Z 1057.326,A -85,B 0,C 180,E1 26536.623,E2 26536.623} C_VEL
LIN {X 0,Y 592.182,Z 1044.233,A -85,B 0,C 180,E1 26535.179,E2 26535.179} C_VEL
LIN {X 0,Y 592.284,Z 1029.578,A -85,B 0,C 180,E1 26533.826,E2 26533.826} C_VEL
LIN {X 0,Y 592.402,Z 1013.883,A -85,B 0,C 180,E1 26532.618,E2 26532.618} C_VEL
LIN {X 0,Y 592.528,Z 997.172,A -85,B 0,C 180,E1 26531.555,E2 26531.555} C_VEL
LIN {X 0,Y 592.651,Z 979.416,A -85,B 0,C 180,E1 26530.639,E2 26530.639} C_VEL
LIN {X 0,Y 592.764,Z 960.822,A -85,B 0,C 180,E1 26529.888,E2 26529.888} C_VEL
LIN {X 0,Y 592.862,Z 941.503,A -85,B 0,C 180,E1 26529.312,E2 26529.312} C_VEL
LIN {X 0,Y 592.936,Z 921.8,A -85,B 0,C 180,E1 26528.922,E2 26528.922} C_VEL
LIN {X 0,Y 593.042,Z 710.776,A -85,B 0,C 180,E1 26526.208,E2 26526.208} C_VEL
LIN {X 0,Y 592.798,Z 708.019,A -85,B 0,C 180,E1 26526.089,E2 26526.089} C_VEL
LIN {X 0,Y 593.06,Z 665.594,A -85,B 0,C 180,E1 26523.139,E2 26523.139} C_VEL
LIN {X 0,Y 593.378,Z 619.648,A -85,B 0,C 180,E1 26519.858,E2 26519.858} C_VEL
LIN {X 0,Y 593.478,Z 605.098,A -85,B 0,C 180,E1 26518.797,E2 26518.797} C_VEL
LIN {X 0,Y 592.039,Z 600.648,A -85,B 0,C 180,E1 26518.34,E2 26518.34} C_VEL
LIN {X 0,Y 592.036,Z 600.489,A -85,B 0,C 180,E1 26515.074,E2 26515.074} C_VEL
LIN {X 0,Y 592.008,Z 600.487,A -85,B 0,C 180,E1 26511.819,E2 26511.819} C_VEL
LIN {X 0,Y 592.026,Z 600.488,A -85,B 0,C 180,E1 26508.673,E2 26508.673} C_VEL
LIN {X 0,Y 592.013,Z 600.487,A -85,B 0,C 180,E1 26505.457,E2 26505.457} C_VEL
LIN {X 0,Y 592.02,Z 600.486,A -85,B 0,C 180,E1 26502.291,E2 26502.291} C_VEL
LIN {X 0,Y 592.02,Z 600.488,A -85,B 0,C 180,E1 26499.172,E2 26499.172} C_VEL
LIN {X 0,Y 592.017,Z 600.485,A -85,B 0,C 180,E1 26495.997,E2 26495.997} C_VEL
LIN {X 0,Y 592.035,Z 600.492,A -85,B 0,C 180,E1 26492.713,E2 26492.713} C_VEL
LIN {X 0,Y 592.033,Z 600.482,A -85,B 0,C 180,E1 26489.372,E2 26489.372} C_VEL
LIN {X 0,Y 592.009,Z 600.49,A -85,B 0,C 180,E1 26486.036,E2 26486.036} C_VEL
LIN {X 0,Y 592.034,Z 600.485,A -85,B 0,C 180,E1 26482.857,E2 26482.857} C_VEL
LIN {X 0,Y 591.997,Z 600.489,A -85,B 0,C 180,E1 26479.742,E2 26479.742} C_VEL
LIN {X 0,Y 592.037,Z 600.487,A -85,B 0,C 180,E1 26476.584,E2 26476.584} C_VEL
LIN {X 0,Y 591.988,Z 600.49,A -85,B 0,C 180,E1 26473.478,E2 26473.478} C_VEL
LIN {X 0,Y 592.038,Z 600.488,A -85,B 0,C 180,E1 26470.312,E2 26470.312} C_VEL
LIN {X 0,Y 591.976,Z 600.492,A -85,B 0,C 180,E1 26467.18,E2 26467.18} C_VEL
LIN {X 0,Y 592.044,Z 600.767,A -85,B 0,C 180,E1 26464.455,E2 26464.455} C_VEL
LIN {X 0,Y 592.642,Z 604.677,A -85,B 0,C 180,E1 26463.966,E2 26463.966} C_VEL
LIN {X 0,Y 592.463,Z 632.758,A -85,B 0,C 180,E1 26460.773,E2 26460.773} C_VEL
LIN {X 0,Y 592.327,Z 662.346,A -85,B 0,C 180,E1 26457.484,E2 26457.484} C_VEL
LIN {X 0,Y 592.209,Z 692.262,A -85,B 0,C 180,E1 26454.234,E2 26454.234} C_VEL
LIN {X 0,Y 592.528,Z 694.921,A -85,B 0,C 180,E1 26454.151,E2 26454.151} C_VEL
LIN {X 0,Y 592.499,Z 722.706,A -85,B 0,C 180,E1 26453.808,E2 26453.808} C_VEL
LIN {X 0,Y 591.554,Z 730.38,A -85,B 0,C 180,E1 26453.74,E2 26453.74} C_VEL
LIN {X 0,Y 585.463,Z 750.727,A -85,B 0,C 180,E1 26453.654,E2 26453.654} C_VEL
LIN {X 0,Y 584.731,Z 757.317,A -85,B 0,C 180,E1 26453.592,E2 26453.592} C_VEL
LIN {X 0,Y 584.646,Z 832.903,A -85,B 0,C 180,E1 26452.624,E2 26452.624} C_VEL
LIN {X 0,Y 584.577,Z 849.902,A -85,B 0,C 180,E1 26452.209,E2 26452.209} C_VEL
LIN {X 0,Y 584.472,Z 865.393,A -85,B 0,C 180,E1 26451.639,E2 26451.639} C_VEL
LIN {X 0,Y 584.363,Z 880.421,A -85,B 0,C 180,E1 26450.888,E2 26450.888} C_VEL
LIN {X 0,Y 584.263,Z 894.252,A -85,B 0,C 180,E1 26449.997,E2 26449.997} C_VEL
LIN {X 0,Y 584.155,Z 907.541,A -85,B 0,C 180,E1 26448.915,E2 26448.915} C_VEL
LIN {X 0,Y 584.072,Z 919.069,A -85,B 0,C 180,E1 26447.744,E2 26447.744} C_VEL
LIN {X 0,Y 584.004,Z 929.406,A -85,B 0,C 180,E1 26446.434,E2 26446.434} C_VEL
LIN {X 0,Y 583.96,Z 938.265,A -85,B 0,C 180,E1 26445.016,E2 26445.016} C_VEL
LIN {X 0,Y 583.933,Z 945.443,A -85,B 0,C 180,E1 26443.513,E2 26443.513} C_VEL
LIN {X 0,Y 583.918,Z 950.901,A -85,B 0,C 180,E1 26441.945,E2 26441.945} C_VEL
LIN {X 0,Y 583.914,Z 954.475,A -85,B 0,C 180,E1 26440.355,E2 26440.355} C_VEL
LIN {X 0,Y 583.913,Z 956.313,A -85,B 0,C 180,E1 26438.673,E2 26438.673} C_VEL
LIN {X 0,Y 583.915,Z 956.227,A -85,B 0,C 180,E1 26437.109,E2 26437.109} C_VEL
LIN {X 0,Y 583.914,Z 954.417,A -85,B 0,C 180,E1 26435.519,E2 26435.519} C_VEL
LIN {X 0,Y 583.918,Z 951.006,A -85,B 0,C 180,E1 26434.001,E2 26434.001} C_VEL
LIN {X 0,Y 583.93,Z 945.714,A -85,B 0,C 180,E1 26432.463,E2 26432.463} C_VEL
LIN {X 0,Y 583.955,Z 938.926,A -85,B 0,C 180,E1 26431.016,E2 26431.016} C_VEL
LIN {X 0,Y 584,Z 930.581,A -85,B 0,C 180,E1 26429.644,E2 26429.644} C_VEL
LIN {X 0,Y 584.062,Z 920.184,A -85,B 0,C 180,E1 26428.294,E2 26428.294} C_VEL
LIN {X 0,Y 584.152,Z 908.416,A -85,B 0,C 180,E1 26427.074,E2 26427.074} C_VEL
LIN {X 0,Y 584.254,Z 895.047,A -85,B 0,C 180,E1 26425.971,E2 26425.971} C_VEL
LIN {X 0,Y 584.364,Z 880.806,A -85,B 0,C 180,E1 26425.043,E2 26425.043} C_VEL
LIN {X 0,Y 584.461,Z 866.339,A -85,B 0,C 180,E1 26424.312,E2 26424.312} C_VEL
LIN {X 0,Y 584.575,Z 850.397,A -85,B 0,C 180,E1 26423.715,E2 26423.715} C_VEL
LIN {X 0,Y 584.642,Z 833.689,A -85,B 0,C 180,E1 26423.301,E2 26423.301} C_VEL
LIN {X 0,Y 584.677,Z 796.327,A -85,B 0,C 180,E1 26422.804,E2 26422.804} C_VEL
LIN {X 0,Y 584.613,Z 694.311,A -85,B 0,C 180,E1 26421.526,E2 26421.526} C_VEL
LIN {X 0,Y 584.358,Z 692.542,A -85,B 0,C 180,E1 26421.477,E2 26421.477} C_VEL
LIN {X 0,Y 584.543,Z 663.537,A -85,B 0,C 180,E1 26418.288,E2 26418.288} C_VEL
LIN {X 0,Y 584.769,Z 632.58,A -85,B 0,C 180,E1 26414.799,E2 26414.799} C_VEL
LIN {X 0,Y 584.968,Z 605.336,A -85,B 0,C 180,E1 26411.673,E2 26411.673} C_VEL
LIN {X 0,Y 584.039,Z 601.567,A -85,B 0,C 180,E1 26411.179,E2 26411.179} C_VEL
LIN {X 0,Y 584.049,Z 601.481,A -85,B 0,C 180,E1 26408.296,E2 26408.296} C_VEL
LIN {X 0,Y 584.036,Z 601.48,A -85,B 0,C 180,E1 26404.996,E2 26404.996} C_VEL
LIN {X 0,Y 584.053,Z 601.48,A -85,B 0,C 180,E1 26402.053,E2 26402.053} C_VEL
LIN {X 0,Y 584.043,Z 601.477,A -85,B 0,C 180,E1 26398.755,E2 26398.755} C_VEL
LIN {X 0,Y 584.061,Z 601.48,A -85,B 0,C 180,E1 26395.774,E2 26395.774} C_VEL
LIN {X 0,Y 584.043,Z 601.478,A -85,B 0,C 180,E1 26392.444,E2 26392.444} C_VEL
LIN {X 0,Y 584.079,Z 601.478,A -85,B 0,C 180,E1 26389.397,E2 26389.397} C_VEL
LIN {X 0,Y 584.046,Z 601.474,A -85,B 0,C 180,E1 26386.176,E2 26386.176} C_VEL
LIN {X 0,Y 584.09,Z 601.482,A -85,B 0,C 180,E1 26383.06,E2 26383.06} C_VEL
LIN {X 0,Y 584.064,Z 601.606,A -85,B 0,C 180,E1 26379.82,E2 26379.82} C_VEL
LIN {X 0,Y 585.098,Z 606.615,A -85,B 0,C 180,E1 26379.145,E2 26379.145} C_VEL
LIN {X 0,Y 584.76,Z 632.807,A -85,B 0,C 180,E1 26376.086,E2 26376.086} C_VEL
LIN {X 0,Y 584.535,Z 660.681,A -85,B 0,C 180,E1 26372.942,E2 26372.942} C_VEL
LIN {X 0,Y 584.371,Z 689.019,A -85,B 0,C 180,E1 26369.804,E2 26369.804} C_VEL
LIN {X 0,Y 584.398,Z 693.041,A -85,B 0,C 180,E1 26369.412,E2 26369.412} C_VEL
LIN {X 0,Y 584.812,Z 698.9,A -85,B 0,C 180,E1 26369.321,E2 26369.321} C_VEL
LIN {X 0,Y 584.643,Z 832.62,A -85,B 0,C 180,E1 26367.63,E2 26367.63} C_VEL
LIN {X 0,Y 584.578,Z 849.587,A -85,B 0,C 180,E1 26367.218,E2 26367.218} C_VEL
LIN {X 0,Y 584.481,Z 864.777,A -85,B 0,C 180,E1 26366.666,E2 26366.666} C_VEL
LIN {X 0,Y 584.37,Z 879.694,A -85,B 0,C 180,E1 26365.928,E2 26365.928} C_VEL
LIN {X 0,Y 584.269,Z 893.638,A -85,B 0,C 180,E1 26365.043,E2 26365.043} C_VEL
LIN {X 0,Y 584.159,Z 906.97,A -85,B 0,C 180,E1 26363.965,E2 26363.965} C_VEL
LIN {X 0,Y 584.077,Z 918.395,A -85,B 0,C 180,E1 26362.821,E2 26362.821} C_VEL
LIN {X 0,Y 584.006,Z 928.69,A -85,B 0,C 180,E1 26361.533,E2 26361.533} C_VEL
LIN {X 0,Y 583.964,Z 937.561,A -85,B 0,C 180,E1 26360.142,E2 26360.142} C_VEL
LIN {X 0,Y 583.936,Z 944.484,A -85,B 0,C 180,E1 26358.744,E2 26358.744} C_VEL
LIN {X 0,Y 583.922,Z 950.007,A -85,B 0,C 180,E1 26357.239,E2 26357.239} C_VEL
LIN {X 0,Y 583.92,Z 954.02,A -85,B 0,C 180,E1 26355.624,E2 26355.624} C_VEL
LIN {X 0,Y 583.915,Z 956.095,A -85,B 0,C 180,E1 26353.997,E2 26353.997} C_VEL
LIN {X 0,Y 583.915,Z 956.37,A -85,B 0,C 180,E1 26352.357,E2 26352.357} C_VEL
LIN {X 0,Y 583.917,Z 954.876,A -85,B 0,C 180,E1 26350.806,E2 26350.806} C_VEL
LIN {X 0,Y 583.922,Z 951.368,A -85,B 0,C 180,E1 26349.136,E2 26349.136} C_VEL
LIN {X 0,Y 583.931,Z 946.326,A -85,B 0,C 180,E1 26347.615,E2 26347.615} C_VEL
LIN {X 0,Y 583.954,Z 939.14,A -85,B 0,C 180,E1 26346.059,E2 26346.059} C_VEL
LIN {X 0,Y 583.999,Z 930.684,A -85,B 0,C 180,E1 26344.658,E2 26344.658} C_VEL
LIN {X 0,Y 584.057,Z 920.5,A -85,B 0,C 180,E1 26343.333,E2 26343.333} C_VEL
LIN {X 0,Y 584.147,Z 909.152,A -85,B 0,C 180,E1 26342.142,E2 26342.142} C_VEL
LIN {X 0,Y 584.246,Z 895.859,A -85,B 0,C 180,E1 26341.033,E2 26341.033} C_VEL
LIN {X 0,Y 584.361,Z 881.789,A -85,B 0,C 180,E1 26340.1,E2 26340.1} C_VEL
LIN {X 0,Y 584.454,Z 867.147,A -85,B 0,C 180,E1 26339.349,E2 26339.349} C_VEL
LIN {X 0,Y 584.565,Z 851.688,A -85,B 0,C 180,E1 26338.756,E2 26338.756} C_VEL
LIN {X 0,Y 584.64,Z 835.589,A -85,B 0,C 180,E1 26338.338,E2 26338.338} C_VEL
LIN {X 0,Y 584.687,Z 812.065,A -85,B 0,C 180,E1 26338,E2 26338} C_VEL
LIN {X 0,Y 584.595,Z 694.207,A -85,B 0,C 180,E1 26336.524,E2 26336.524} C_VEL
LIN {X 0,Y 584.363,Z 692.113,A -85,B 0,C 180,E1 26336.437,E2 26336.437} C_VEL
LIN {X 0,Y 584.534,Z 662.973,A -85,B 0,C 180,E1 26333.225,E2 26333.225} C_VEL
LIN {X 0,Y 584.761,Z 633.9,A -85,B 0,C 180,E1 26329.949,E2 26329.949} C_VEL
LIN {X 0,Y 585.109,Z 607.074,A -85,B 0,C 180,E1 26326.813,E2 26326.813} C_VEL
LIN {X 0,Y 584.553,Z 603.432,A -85,B 0,C 180,E1 26326.347,E2 26326.347} C_VEL
LIN {X 0,Y 584.114,Z 601.579,A -85,B 0,C 180,E1 26326.047,E2 26326.047} C_VEL
LIN {X 0,Y 584.09,Z 601.482,A -85,B 0,C 180,E1 26322.679,E2 26322.679} C_VEL
LIN {X 0,Y 584.082,Z 601.474,A -85,B 0,C 180,E1 26319.427,E2 26319.427} C_VEL
LIN {X 0,Y 584.081,Z 601.477,A -85,B 0,C 180,E1 26316.199,E2 26316.199} C_VEL
LIN {X 0,Y 584.079,Z 601.476,A -85,B 0,C 180,E1 26312.982,E2 26312.982} C_VEL
LIN {X 0,Y 584.078,Z 601.475,A -85,B 0,C 180,E1 26309.765,E2 26309.765} C_VEL
LIN {X 0,Y 584.083,Z 601.478,A -85,B 0,C 180,E1 26306.538,E2 26306.538} C_VEL
LIN {X 0,Y 584.084,Z 601.473,A -85,B 0,C 180,E1 26303.293,E2 26303.293} C_VEL
LIN {X 0,Y 584.095,Z 601.482,A -85,B 0,C 180,E1 26299.985,E2 26299.985} C_VEL
LIN {X 0,Y 584.093,Z 601.472,A -85,B 0,C 180,E1 26296.611,E2 26296.611} C_VEL
LIN {X 0,Y 584.08,Z 601.478,A -85,B 0,C 180,E1 26293.362,E2 26293.362} C_VEL
LIN {X 0,Y 584.086,Z 601.472,A -85,B 0,C 180,E1 26290.156,E2 26290.156} C_VEL
LIN {X 0,Y 584.075,Z 601.476,A -85,B 0,C 180,E1 26286.981,E2 26286.981} C_VEL
LIN {X 0,Y 584.085,Z 601.474,A -85,B 0,C 180,E1 26283.828,E2 26283.828} C_VEL
LIN {X 0,Y 584.072,Z 601.474,A -85,B 0,C 180,E1 26280.589,E2 26280.589} C_VEL
LIN {X 0,Y 584.086,Z 601.476,A -85,B 0,C 180,E1 26277.449,E2 26277.449} C_VEL
LIN {X 0,Y 584.072,Z 601.475,A -85,B 0,C 180,E1 26274.302,E2 26274.302} C_VEL
LIN {X 0,Y 584.087,Z 601.475,A -85,B 0,C 180,E1 26271.138,E2 26271.138} C_VEL
LIN {X 0,Y 584.07,Z 601.475,A -85,B 0,C 180,E1 26267.945,E2 26267.945} C_VEL
LIN {X 0,Y 584.09,Z 601.477,A -85,B 0,C 180,E1 26264.715,E2 26264.715} C_VEL
LIN {X 0,Y 584.076,Z 601.471,A -85,B 0,C 180,E1 26261.508,E2 26261.508} C_VEL
LIN {X 0,Y 584.097,Z 601.48,A -85,B 0,C 180,E1 26258.194,E2 26258.194} C_VEL
LIN {X 0,Y 584.098,Z 601.471,A -85,B 0,C 180,E1 26254.879,E2 26254.879} C_VEL
LIN {X 0,Y 584.071,Z 601.478,A -85,B 0,C 180,E1 26251.582,E2 26251.582} C_VEL
LIN {X 0,Y 584.093,Z 601.471,A -85,B 0,C 180,E1 26248.412,E2 26248.412} C_VEL
LIN {X 0,Y 584.067,Z 601.477,A -85,B 0,C 180,E1 26245.246,E2 26245.246} C_VEL
LIN {X 0,Y 584.093,Z 601.474,A -85,B 0,C 180,E1 26242.081,E2 26242.081} C_VEL
LIN {X 0,Y 584.064,Z 601.477,A -85,B 0,C 180,E1 26238.871,E2 26238.871} C_VEL
LIN {X 0,Y 584.092,Z 601.475,A -85,B 0,C 180,E1 26235.687,E2 26235.687} C_VEL
LIN {X 0,Y 584.061,Z 601.477,A -85,B 0,C 180,E1 26232.547,E2 26232.547} C_VEL
LIN {X 0,Y 584.091,Z 601.477,A -85,B 0,C 180,E1 26229.426,E2 26229.426} C_VEL
LIN {X 0,Y 584.06,Z 601.479,A -85,B 0,C 180,E1 26226.263,E2 26226.263} C_VEL
LIN {X 0,Y 584.093,Z 601.478,A -85,B 0,C 180,E1 26223.097,E2 26223.097} C_VEL
LIN {X 0,Y 584.095,Z 601.726,A -85,B 0,C 180,E1 26222.05,E2 26222.05} C_VEL
